// TwinCAT 3 PLC project Core
// ProgramVersion: 3.1.4023.0
// libraries:
//   CmpBitmapPool, * (System)
//   Tc2_MC2, * (Beckhoff Automation GmbH)
//   Tc2_MDP, * (Beckhoff Automation GmbH)
//   Tc2_Standard, * (Beckhoff Automation GmbH)
//   Tc2_System, * (Beckhoff Automation GmbH)
//   Tc2_Utilities, * (Beckhoff Automation GmbH)
//   Tc3_IotBase, * (Beckhoff Automation GmbH)
//   Tc3_Module, * (Beckhoff Automation GmbH)
//   VisuDialogs, * (System)
// project tree:
//   DUTs/ E_Balise.TcDUT, E_Type_motion.TcDUT, E_Type_Tache.TcDUT, ST_Dynamixel_Control_Input.TcDUT, ST_Dynamixel_Control_Output.TcDUT, ST_Tableau.TcDUT
//   / GlobalTextList.TcGTLO
//   GVLs/Action/ G_CAM.TcGVL, G_DXL.TcGVL
//   GVLs/Interruption/ G_Balise.TcGVL
//   GVLs/IO/ G_IO.TcGVL
//   GVLs/Motion/ G_Moteurs.TcGVL, G_Odometrie.TcGVL
//   GVLs/Raspberry PI/ G_RPI.TcGVL
//   GVLs/Structure/ G_EndMatch.TcGVL, G_init.TcGVL, G_Match.TcGVL, G_PreMatch.TcGVL
//   GVLs/Visu/ G_Visus.TcGVL
//   POUs/Action/Camera OAK-D/ FB_CAM.TcPOU, P_cam_launch_pyscript.TcPOU
//   POUs/Action/Dynamixel/ FB_DXL_AX12A.TcPOU, FB_DXL_XL.TcPOU, P_Connect_DXL.TcPOU, P_DXL_launch_pyscript.TcPOU
//   POUs/Action/ ITAction.TcPOU
//   POUs/Communication/ ITCommunication.TcPOU, MQTT.TcPOU
//   POUs/Interruption/ FB_Balise.TcPOU, FB_Timeout.TcPOU, ITInterruption.TcPOU
//   POUs/ MAIN.TcPOU
//   POUs/Motion/ FB_Motion_Odometrie.TcPOU, ITMotion.TcPOU
//   POUs/Structure/Actions/ F_DXL_Position.TcPOU, F_DXL_Reset.TcPOU
//   POUs/Structure/ Structure_MAIN.TcPOU
//   POUs/Structure/Tableaux %28parcours%29/ P_Tableau_Strategie_1.TcPOU (not stored), P_Tableau_Strategie_2.TcPOU (not stored)
//   POUs/Utillity/Debug/ pass.TcPOU (not stored)
//   POUs/Utillity/Logic/ plusOuMoins.TcPOU
//   POUs/Utillity/Maths/ DEGRE2RAD.TcPOU, HYP.TcPOU, RAD2DEGRE.TcPOU
//   POUs/Utillity/Structure/Action/ FinishAction.TcPOU, Next.TcPOU (not stored), StartAction.TcPOU (not stored)
//   POUs/Utillity/Structure/Tableau/ AddStep.TcPOU, EtapeEnCours.TcPOU (not stored), PointsRestants.TcPOU, ReplaceStep.TcPOU
//   POUs/Utillity/Temporisation/ delay.TcPOU
//   TASKs/ BaliseTask.TcTTO, MotionTask.TcTTO, PlcTask.TcTTO, VISU_TASK.TcTTO
//   VISUs/Visu pour debug/ V_Balise.TcVIS, V_Config.TcVIS, V_Deplacement.TcVIS, V_Test.TcVIS
//   VISUs/Images/ ImagePool.TcIPO (not stored)
//   VISUs/Visu pour match/ V_Fin_Match.TcVIS, V_Init.TcVIS, V_Match.TcVIS
//   VISUs/ VisualizationManager.TcVMO (not stored), V_Menu.TcVIS
// real-time tasks:
//   TASK PlcTask: cycle T#10ms, priority 20, ADS port 350
//   TASK VisuTask: cycle T#100000us, priority 30, ADS port 351
//   TASK BaliseTask: cycle T#1ms, priority 5, ADS port 352
//   TASK MotionTask: cycle T#5ms, priority 15, ADS port 353
// motion (NC):
//   TASK NC-Task 1 SAF: cycle T#1ms, priority 4, ADS port 501
//   TASK NC-Task 1 SVB: cycle T#5ms, priority 8, ADS port 511
//   AXIS MoteurG (id 1)
//     Dynamic: Acceleration=3000, Deceleration=3000, Jerk=9000, MaxPosDeviationAuxAxis=5
//     Velo: SlowManual=200
//     PositionAreaControl: Range=10
//     TargetPosControl: Range=10
//     OtherSettings: AllowMotionCmdToSlave=true
//     encoder EncType=4
//       EncPara: ScaleFactorNumerator=162, ScaleFactorDenominator=12800, MaxCount=#x0000ffff
//         ActPosCorrection: Enable=true
//         Inc: RefSoftSyncMask=#x0000ffff
//     drive DrvType=24
//       Analog: VeloReferenz=1700, TorqueSetpointScale=10, ScaleFactorActTorque=0.1
//       TimeComp: TaskDelayCycles=1
//     controller CtrType=1
//       CtrPara: PriorControlFactor=1
//         PosDiffControl: Enable=false, Range=20
//         Observer: BandWidth=20
//   AXIS EncodeurG (id 3)
//     OtherSettings: AllowMotionCmdToSlave=true
//     encoder EncType=4
//       EncPara: ScaleFactorNumerator=162, ScaleFactorDenominator=4096, MaxCount=#x0000ffff
//         Inc: RefSoftSyncMask=#x0000ffff
//     drive DrvType=5
//       Analog: TorqueSetpointScale=10, ScaleFactorActTorque=0.1
//       TimeComp: TaskDelayCycles=1
//     controller CtrType=1
//       CtrPara: PriorControlFactor=1
//         Observer: BandWidth=20
//   AXIS MoteurD (id 2)
//     Dynamic: Acceleration=3000, Deceleration=3000, Jerk=9000, MaxPosDeviationAuxAxis=5
//     Velo: SlowManual=200
//     PositionAreaControl: Range=10
//     TargetPosControl: Range=10
//     OtherSettings: AllowMotionCmdToSlave=true
//     encoder EncType=4
//       EncPara: ScaleFactorNumerator=162, ScaleFactorDenominator=12800, MaxCount=#x0000ffff
//         Inc: RefSoftSyncMask=#x0000ffff
//     drive DrvType=24
//       Analog: VeloReferenz=1700, TorqueSetpointScale=10, ScaleFactorActTorque=0.1
//       TimeComp: TaskDelayCycles=1
//     controller CtrType=1
//       CtrPara: PriorControlFactor=1
//         PosDiffControl: Enable=false, Range=20
//         Observer: BandWidth=20
//   AXIS EncodeurD (id 4)
//     OtherSettings: AllowMotionCmdToSlave=true
//     encoder EncType=4
//       EncPara: ScaleFactorNumerator=162, ScaleFactorDenominator=4096, MaxCount=#x0000ffff
//         Inc: RefSoftSyncMask=#x0000ffff
//     drive DrvType=5
//       Analog: TorqueSetpointScale=10, ScaleFactorActTorque=0.1
//       TimeComp: TaskDelayCycles=1
//     controller CtrType=1
//       CtrPara: PriorControlFactor=1
//         Observer: BandWidth=20
// I/O:
//   DEVICE Device 3 (EtherCAT), AmsNetId 172.16.0.209.4.1
//     Term 1 (EK1100) [EK1100 EtherCAT Coupler (2A E-Bus)]
//       T_Balise (EL1252) [EL1252 2Ch. Fast Dig. Input 24V, 1µs, DC Latch]
//       T_Input (EL1104) [EL1104 4Ch. Dig. Input 24V, 3ms, Sensor Power]
//       T_MoteurG (EL7037) [EL7037 1Ch. Stepper motor output stage (24V, 1.5A)]
//       T_MoteurD (EL7037) [EL7037 1Ch. Stepper motor output stage (24V, 1.5A)]
//       T_Output (EL2798) [EL2798 8Ch. Dig. Output 24V AC/DC, 2A, potential-free]
//       Term 5 (EL9011) [EL9011 End Terminal]
// variable links:
//   NC-Task 1 SAF/Axes/EncodeurD <-> Device 3 (EtherCAT)/Term 1 (EK1100)/T_MoteurD (EL7037)
//     Enc/Inputs/In/nDataIn1 <-> STM External position/External position
//     Enc/Inputs/In/nState4 @bit 1 <-> WcState/InputToggle
//     Enc/Inputs/In/nState4 <-> WcState/WcState
//   NC-Task 1 SAF/Axes/EncodeurG <-> Device 3 (EtherCAT)/Term 1 (EK1100)/T_MoteurG (EL7037)
//     Enc/Inputs/In/nDataIn1 <-> STM External position/External position
//     Enc/Inputs/In/nState4 @bit 1 <-> WcState/InputToggle
//     Enc/Inputs/In/nState4 <-> WcState/WcState
//   NC-Task 1 SAF/Axes/MoteurD <-> Device 3 (EtherCAT)/Term 1 (EK1100)/T_MoteurD (EL7037)
//     Drive/Inputs/In/nState1 @bit 3 <-> STM Status/Error
//     Drive/Inputs/In/nState1 @bit 7 <-> STM Status/Motor stall
//     Drive/Inputs/In/nState1 @bit 5 <-> STM Status/Moving negative
//     Drive/Inputs/In/nState1 @bit 4 <-> STM Status/Moving positive
//     Drive/Inputs/In/nState1 @bit 1 <-> STM Status/Ready
//     Drive/Inputs/In/nState1 <-> STM Status/Ready to enable
//     Drive/Inputs/In/nState1 @bit 6 <-> STM Status/Torque reduced
//     Drive/Inputs/In/nState1 @bit 2 <-> STM Status/Warning
//     Drive/Inputs/In/nState2 @bit 3 <-> STM Status/Digital input 1
//     Drive/Inputs/In/nState2 @bit 4 <-> STM Status/Digital input 2
//     Drive/Inputs/In/nState2 @bit 5 <-> STM Status/Sync error
//     Drive/Inputs/In/nState2 @bit 7 <-> STM Status/TxPDO Toggle
//     Drive/Inputs/In/nState4 @bit 1 <-> WcState/InputToggle
//     Drive/Inputs/In/nState4 <-> WcState/WcState
//     Drive/Outputs/Out/nCtrl1 <-> STM Control/Enable
//     Drive/Outputs/Out/nCtrl1 @bit 2 <-> STM Control/Reduce torque
//     Drive/Outputs/Out/nCtrl1 @bit 1 <-> STM Control/Reset
//     Drive/Outputs/Out/nCtrl2 @bit 3 <-> STM Control/Digital output 1
//     Drive/Outputs/Out/nDataOut2[0] <-> STM Velocity/Velocity
//     Enc/Inputs/In/nDataIn1[0] <-> ENC Status compact/Counter value
//     Enc/Inputs/In/nDataIn2[0] <-> ENC Status compact/Latch value
//     Enc/Inputs/In/nState1 @bit 4 <-> ENC Status compact/Counter overflow
//     Enc/Inputs/In/nState1 @bit 3 <-> ENC Status compact/Counter underflow
//     Enc/Inputs/In/nState1 @bit 7 <-> ENC Status compact/Extrapolation stall
//     Enc/Inputs/In/nState1 <-> ENC Status compact/Latch C valid
//     Enc/Inputs/In/nState1 @bit 1 <-> ENC Status compact/Latch extern valid
//     Enc/Inputs/In/nState1 @bit 2 <-> ENC Status compact/Set counter done
//     Enc/Inputs/In/nState2 @bit 4 <-> ENC Status compact/Status of extern latch
//     Enc/Inputs/In/nState2 <-> ENC Status compact/Status of input A
//     Enc/Inputs/In/nState2 @bit 1 <-> ENC Status compact/Status of input B
//     Enc/Inputs/In/nState2 @bit 2 <-> ENC Status compact/Status of input C
//     Enc/Inputs/In/nState2 @bit 5 <-> ENC Status compact/Sync error
//     Enc/Inputs/In/nState2 @bit 7 <-> ENC Status compact/TxPDO Toggle
//     Enc/Inputs/In/nState4 @bit 1 <-> WcState/InputToggle
//     Enc/Inputs/In/nState4 <-> WcState/WcState
//     Enc/Outputs/Out/nCtrl1 <-> ENC Control compact/Enable latch C
//     Enc/Outputs/Out/nCtrl1 @bit 3 <-> ENC Control compact/Enable latch extern on negative edge
//     Enc/Outputs/Out/nCtrl1 @bit 1 <-> ENC Control compact/Enable latch extern on positive edge
//     Enc/Outputs/Out/nCtrl1 @bit 2 <-> ENC Control compact/Set counter
//     Enc/Outputs/Out/nDataOut1[0] <-> ENC Control compact/Set counter value
//   NC-Task 1 SAF/Axes/MoteurG <-> Device 3 (EtherCAT)/Term 1 (EK1100)/T_MoteurG (EL7037)
//     Drive/Inputs/In/nState1 @bit 3 <-> STM Status/Error
//     Drive/Inputs/In/nState1 @bit 7 <-> STM Status/Motor stall
//     Drive/Inputs/In/nState1 @bit 5 <-> STM Status/Moving negative
//     Drive/Inputs/In/nState1 @bit 4 <-> STM Status/Moving positive
//     Drive/Inputs/In/nState1 @bit 1 <-> STM Status/Ready
//     Drive/Inputs/In/nState1 <-> STM Status/Ready to enable
//     Drive/Inputs/In/nState1 @bit 6 <-> STM Status/Torque reduced
//     Drive/Inputs/In/nState1 @bit 2 <-> STM Status/Warning
//     Drive/Inputs/In/nState2 @bit 3 <-> STM Status/Digital input 1
//     Drive/Inputs/In/nState2 @bit 4 <-> STM Status/Digital input 2
//     Drive/Inputs/In/nState2 @bit 5 <-> STM Status/Sync error
//     Drive/Inputs/In/nState2 @bit 7 <-> STM Status/TxPDO Toggle
//     Drive/Inputs/In/nState4 @bit 1 <-> WcState/InputToggle
//     Drive/Inputs/In/nState4 <-> WcState/WcState
//     Drive/Outputs/Out/nCtrl1 <-> STM Control/Enable
//     Drive/Outputs/Out/nCtrl1 @bit 2 <-> STM Control/Reduce torque
//     Drive/Outputs/Out/nCtrl1 @bit 1 <-> STM Control/Reset
//     Drive/Outputs/Out/nCtrl2 @bit 3 <-> STM Control/Digital output 1
//     Drive/Outputs/Out/nDataOut2[0] <-> STM Velocity/Velocity
//     Enc/Inputs/In/nDataIn1[0] <-> ENC Status compact/Counter value
//     Enc/Inputs/In/nDataIn2[0] <-> ENC Status compact/Latch value
//     Enc/Inputs/In/nState1 @bit 4 <-> ENC Status compact/Counter overflow
//     Enc/Inputs/In/nState1 @bit 3 <-> ENC Status compact/Counter underflow
//     Enc/Inputs/In/nState1 @bit 7 <-> ENC Status compact/Extrapolation stall
//     Enc/Inputs/In/nState1 <-> ENC Status compact/Latch C valid
//     Enc/Inputs/In/nState1 @bit 1 <-> ENC Status compact/Latch extern valid
//     Enc/Inputs/In/nState1 @bit 2 <-> ENC Status compact/Set counter done
//     Enc/Inputs/In/nState2 @bit 4 <-> ENC Status compact/Status of extern latch
//     Enc/Inputs/In/nState2 <-> ENC Status compact/Status of input A
//     Enc/Inputs/In/nState2 @bit 1 <-> ENC Status compact/Status of input B
//     Enc/Inputs/In/nState2 @bit 2 <-> ENC Status compact/Status of input C
//     Enc/Inputs/In/nState2 @bit 5 <-> ENC Status compact/Sync error
//     Enc/Inputs/In/nState2 @bit 7 <-> ENC Status compact/TxPDO Toggle
//     Enc/Inputs/In/nState4 @bit 1 <-> WcState/InputToggle
//     Enc/Inputs/In/nState4 <-> WcState/WcState
//     Enc/Outputs/Out/nCtrl1 <-> ENC Control compact/Enable latch C
//     Enc/Outputs/Out/nCtrl1 @bit 3 <-> ENC Control compact/Enable latch extern on negative edge
//     Enc/Outputs/Out/nCtrl1 @bit 1 <-> ENC Control compact/Enable latch extern on positive edge
//     Enc/Outputs/Out/nCtrl1 @bit 2 <-> ENC Control compact/Set counter
//     Enc/Outputs/Out/nDataOut1[0] <-> ENC Control compact/Set counter value
//   Core/Core Instance <-> Device 3 (EtherCAT)/Term 1 (EK1100)/T_Balise (EL1252)
//     BaliseTask Inputs/G_Balise.Inductif <-> Channel 1/Input
//     BaliseTask Inputs/G_Balise.Laser <-> Channel 2/Input
//     BaliseTask Inputs/ITInterruption.balise.DebutDetection <-> Latch/LatchNeg2
//     BaliseTask Inputs/ITInterruption.balise.DebutTour <-> Latch/LatchPos1
//     BaliseTask Inputs/ITInterruption.balise.FinDetection <-> Latch/LatchPos2
//   Core/Core Instance <-> Device 3 (EtherCAT)/Term 1 (EK1100)/T_Input (EL1104)
//     BaliseTask Inputs/G_IO.bAU <-> Channel 1/Input
//     PlcTask Inputs/G_IO.bCaptDepart <-> Channel 2/Input
//   Core/Core Instance <-> Device 3 (EtherCAT)/Term 1 (EK1100)/T_Output (EL2798)
//     BaliseTask Outputs/G_IO.bMoteurBalise <-> Channel 1/Output
//     PlcTask Outputs/G_IO.bLEDInit <-> Channel 2/Output
//   Core/Core Instance <-> NC-Task 1 SAF/Axes/EncodeurD
//     BaliseTask Inputs/G_Moteurs.axEncodeurD.NcToPlc <-> Outputs/ToPlc
//     MotionTask Outputs/G_Moteurs.axEncodeurD.PlcToNc <-> Inputs/FromPlc
//   Core/Core Instance <-> NC-Task 1 SAF/Axes/EncodeurG
//     MotionTask Inputs/G_Moteurs.axEncodeurG.NcToPlc <-> Outputs/ToPlc
//     MotionTask Outputs/G_Moteurs.axEncodeurG.PlcToNc <-> Inputs/FromPlc
//   Core/Core Instance <-> NC-Task 1 SAF/Axes/MoteurD
//     MotionTask Inputs/G_Moteurs.axMoteurD.NcToPlc <-> Outputs/ToPlc
//     MotionTask Outputs/G_Moteurs.axMoteurD.PlcToNc <-> Inputs/FromPlc
//   Core/Core Instance <-> NC-Task 1 SAF/Axes/MoteurG
//     MotionTask Inputs/G_Moteurs.axMoteurG.NcToPlc <-> Outputs/ToPlc
//     MotionTask Outputs/G_Moteurs.axMoteurG.PlcToNc <-> Inputs/FromPlc

CONFIGURATION Core
    RESOURCE PLC ON TwinCAT3
        TASK BaliseTask(INTERVAL := T#1ms, PRIORITY := 5);
        TASK MotionTask(INTERVAL := T#5ms, PRIORITY := 15);
        TASK PlcTask(INTERVAL := T#10ms, PRIORITY := 20);
        TASK VISU_TASK(INTERVAL := T#100000us, PRIORITY := 30);
        PROGRAM ITInterruption WITH BaliseTask : ITInterruption;
        PROGRAM ITMotion WITH MotionTask : ITMotion;
        PROGRAM MAIN WITH PlcTask : MAIN;
        PROGRAM VisuElems_Visu_Prg WITH VISU_TASK : VisuElems.Visu_Prg;
    END_RESOURCE
END_CONFIGURATION

// ---- DUTs/E_Balise.TcDUT
{attribute 'qualified_only'}
{attribute 'strict'}
TYPE E_Balise :
(
	Angle, Distance
);
END_TYPE

// ---- DUTs/E_Type_motion.TcDUT
TYPE E_Type_motion :
(
	eCoordonne, eMarcheArriereCoordonne, eDistance, eAngle, eCourbe 
);
END_TYPE

// ---- DUTs/E_Type_Tache.TcDUT
TYPE E_Type_Tache :	// Appel des différentes tâches que le robot va faire
(
	eAttendre, eDeplacement, eAction, eFinParcours, eChangementTache
);
END_TYPE

// ---- DUTs/ST_Dynamixel_Control_Input.TcDUT
TYPE ST_Dynamixel_Control_Input :
	STRUCT	
		TypeAX : FB_DXL_AX12A;
		TypeXL : FB_DXL_XL;
		
		bEnableTorque : BOOL;
		bDisableTorque: BOOL;
		
		bLedOn : BOOL;
		IbLedOff : BOOL;
		
		bOperatingMode : BOOL;
		
		bPosition : BOOL;
		bStopPosition : BOOL;
		bResetPosition : BOOL;
		bAcceleration : BOOL;
		bVelocity : BOOL;
		
		ParamOperatingMode_string : STRING;
		ParamReset_BOOL : BOOL;
		ParamPosition_DINT : DINT;
		ParamSpeed_INT : INT;
		ParamAcceleration_USINT : USINT;
		
		bGetLoad : BOOL;
		bGetMovement : BOOL;
		bGetPosition : BOOL;
	END_STRUCT
END_TYPE

// ---- DUTs/ST_Dynamixel_Control_Output.TcDUT
TYPE ST_Dynamixel_Control_Output :
	STRUCT	
		bEnableTorque : BOOL;
		bDisableTorque: BOOL;
		
		bLedOn : BOOL;
		bLedOff : BOOL;
		
		bOperatingMode : BOOL;
		
		bPosition : BOOL;
		bStopPosition : BOOL;
		bResetPosition : BOOL;
		bAcceleration : BOOL;
		bVelocity : BOOL;

		INFO_load_int :INT := -9000;
		INFO_Mouvement_bool : BOOL := 1;
		INFO_Position_dint : DINT := -9000;
	END_STRUCT
END_TYPE

// ---- DUTs/ST_Tableau.TcDUT
TYPE ST_Tableau : // Appel des variables qui permettent de faire les différentes tâches
	STRUCT
		NomEtape			: STRING(50);			// Nom de l'étape en cours => permet de faire des saut dans le tableau pour cibler une action en particulier
		EtapeCible			: STRING(50); 			// Nom de l'étape à laquelle on veut aller
		TypeTache			: E_Type_Tache;			// Permet la tâche qu'on va faire à la ligne du tableau
		TypeDeplacement     : E_Type_motion;        // Permet de choisir le type de déplacement
		TypeAction			: STRING(50);			// Choisi le type d'action
		lrPositionX_mm		: LREAL;				// Position en x que l'on veut donner au robot lors d'un déplacement
		lrPositionY_mm		: LREAL;				// Position en y que le robot doit atteindre lors d'un déplacement
		lrAngleVoulu_deg	: LREAL;				// Angle que l'on veut atteindre lors d'une rotation, en fonction de l'angle de référence dans Odometrie
		lrDistanceVoulu_mm	: LREAL;				// Distance que le robot va avancer
		lrVitesse_mms		: LREAL;				// Vitesse de déplacement du robot quand il fait un mouvement ou une rotation
		lrRayonCourbe_mm	: LREAL;
		tAttente_ms			: TIME;					// Temps que le robot va attendre quand la tâche attente est choisie
		uiAjoutPoints_pts	: INT;					// Nombre de points que l'on veut ajouter sur le compteur
		bArretDetection		: BOOL;					// Désactivation de la détection de la balise, le robot ne s'arrête plus quand il détecte un adversaire, sert à pouvoir démarrer si nos robots ont aussi des catadioptres
	END_STRUCT
END_TYPE

// ---- GVLs/Action/G_CAM.TcGVL
{attribute 'qualified_only'}
//author: Alec Horth

// servent à la communication PYADS (! ne pas modifier)
//seulement accessible au FB "FB_CAM"
VAR_GLOBAL
	//RUN variable => active les fonctionnalités de la caméra
	//sinon les fonctions ne sont pas active pour economiser les ressources de la CPU (!! garde la dernière valeur)
	RUN_STEREO			:BOOL; //mesure de proximité
	RUN_ARUCO			:BOOL; //liste les ID des tags aruco présents dans le champ de vision de la caméra
	
	//retour de la caméra 
	proximite			:USINT; //mesure de proximité de 0 à 3 
							   //(0:champ de vision vide, 1:objet détecté, 2:object proche, 3:distance critique)
	tag_aruco			:ARRAY[0..10] OF INT; //list les id des tags aruco présent 
											  // max 10 tag détectés en même temps (défini par la longeur max de la liste)
	taille_tag_aruco_cm :INT;
	ID_tag_aruco		:INT;
	
	//fonctions du script python
	STOP_PYSCRIPT		:BOOL; //arrête le script python
	restart_py_script	:BOOL:= FALSE; //démarre le script python
	bPyscript_running	:BOOL;		//le script python est actif
END_VAR

// ---- GVLs/Action/G_DXL.TcGVL
{attribute 'qualified_only'}
//author: Alec Horth

//servent à la communication PYADS (! ne pas modifier)
//seulement accessible au FB "FB_DXL_ALL"
VAR_GLOBAL 
	//activation des fonction du moteur dynamixel
	bRun					:BOOL;		// action la fonction
	bStop_python_script		:BOOL; 		// arrête le script python
	
	//commande envoyé au moteur 
	iID						:INT;		// id du motor 
	usiMotor_type			:USINT;		// type du moteur 1 => AX12A, 2 => XL430
	usiFonction 			:USINT;		// fonction à executer
	sMode					:STRING;	// configuration du mode de fonctionnement (position, velocité)
	iSpeed					:INT;		// configuration de la vitesse
	diPosition				:DINT;		// configuration de la position
	usiAcceleration			:USINT; 	// configuration de l'accelération du moteur
	bReset					:BOOL;		// reset de la position en mode multitour
	
	//information du moteur
	iDxl_load				:INT; 
	diDxl_position			:DINT;
	bDxl_movement			:BOOL;
	bDone					:BOOL;		//action reçue et envoyée
	bPyscript_running		:BOOL;		//le script python est actif
	
	// semaphore (contrôle qu'il n'y aie qu'une communication à la fois avec le moteur)
	// indique l'ID de l'instance qui a le droit de communiquer avec le moteur
	// Token disponible => -16#FE ou -254 ou -1 * id_du_moteur_ayant_la_permission
	bToken					:INT:= -16#FE; 
	
	//activation du script python
	bRestart_py_script		:BOOL;
END_VAR

//type de commandes à envoyer au moteur
VAR_GLOBAL CONSTANT 
	//RAM
	usiOPERATING_MODE		:USINT := 0;
	
	//ACTION
	usiENABLE_TORQUE		:USINT := 1; 
	usiDISABLE_TORQUE		:USINT := 2;
	usiLED_ON				:USINT := 3;
	usiLED_OFF				:USINT := 4;
	usiGOAL_ACCELERATION	:USINT := 5;
	usiGOAL_VELOCITY		:USINT := 6;
	usiGOAL_POSITION		:USINT := 7;
	
	//prédicat
	usiGET_PRESENT_POSITION:USINT := 8;
    usiGET_PRESENT_LOAD	:USINT := 9;
    usiGET_PRESENT_MOVEMENT:USINT := 10;
	
	//fonction accessoire du mode position
	usiSTOP_POSITION		:USINT := 11;
	usiRESET_POSITION		:USINT := 12;
	
	//token libre
	iOPEN_TOKEN			:INT   := -254;
END_VAR

// ---- GVLs/Interruption/G_Balise.TcGVL
{attribute 'qualified_only'}
VAR_GLOBAL
	Laser 				AT%I* 	: BOOL; 			//capteur optique de proximité (avec le mirroir)
	Inductif 			AT%I* 	: BOOL; 			//capteur induction sous la balise	
	
	iNombreEnnemi 				: INT;				// nombre de fronts montants du laser, nombres d'ennemis détectés en un tour
	ArrayEnnemi					: ARRAY [0..2,0..1] OF LREAL; 	// 	colonnes = ennemis 	[colonne, ligne]
																//	ligne 0 = Angle 	[colonne, ligne]
                                                        		// 	ligne 1 = Distance 	[colonne, ligne]
	
	bFront 						: BOOL;				//adversaire devant
	bBack 						: BOOL;				//adversaire derrière
	bLeft						: BOOL;				//adversaire à gauche
	bRight						: BOOL;				//adversaire à droite
	bProche						: BOOL;				//obstacle détecté proche
	bClose 						: BOOL;				//obstacle détecté vraiment proche	
	
	lrDistance_1				: LREAL;			// Distance du premier ennemi détecté, est envoyée dans la visu balise
	lrDistance_2				: LREAL;			// Distance du deuxième adversaire détecté, est envoyée dans la visu balise
	lrDistance_3				: LREAL;			// Distance du troisième ennemi détecté, est envoyée dans la visu balise
	lrAngle_1					: LREAL;			// Angle auquel le premier ennemi est détecté pour pouvoir le voir dans la visu balise
	lrAngle_2					: LREAL;			// Angle de détection du deuxième adversaire, l'angle est envoyé dans la visu balise
	lrAngle_3					: LREAL;			// Angle du troisième adversaire , permet de savoir la position de l'ennemi dans la visu balise

	lrCoord_X1					: LREAL;			//coordonné X de l'enemi 1 selon le système de l'odométrie (activé avec la visu)
	lrCoord_Y1					: LREAL;			//coordonné Y de l'enemi 1 selon le système de l'odométrie (activé avec la visu)
	lrCoord_X2					: LREAL; 			//coordonné X de l'enemi 2 selon le système de l'odométrie (activé avec la visu)
	lrCoord_Y2					: LREAL; 			//coordonné Y de l'enemi 2 selon le système de l'odométrie (activé avec la visu)
	lrCoord_X3					: LREAL;			//coordonné X de l'enemi 3 selon le système de l'odométrie (activé avec la visu)
	lrCoord_Y3					: LREAL;			//coordonné Y de l'enemi 3 selon le système de l'odométrie (activé avec la visu)
END_VAR

// ---- GVLs/IO/G_IO.TcGVL
{attribute 'qualified_only'}
VAR_GLOBAL
	// Variable en cas de panneau de commande sur le robot, sinon remplacer par des boutons visus.
	bAU				AT%I*: BOOL;	// Bouton d'arrêt d'urgence, contact NC
	bChoixCote		AT%I*: BOOL;	// Selecteur deux positions pour le choix du coté de départ (jaune=true, violet=false)
	bInitRobot		AT%I*: BOOL;	// Bouton poussoir pour l'initialisation du robot, action et position
	bCaptDepart		AT%I*: BOOL;	// Capteur inductif pour commencer un match
	bReset			AT%I*: BOOL;	// Redémarre Twincat
	
	bLEDInit		AT%Q*: BOOL;	// LED robot initialisé, s'allume quand le robot est initialisé
	bMoteurBalise	AT%Q*: BOOL;	// Moteur de la balise, fait tourner le rayon pour détecter les adversaires
END_VAR

// ---- GVLs/Motion/G_Moteurs.TcGVL
{attribute 'qualified_only'}
VAR_GLOBAL
	axMoteurG		: AXIS_REF;			// Moteur gauche de la base roulante
	axMoteurD		: AXIS_REF;			// Moteur droit de la base roulante
	axEncodeurG		: AXIS_REF;			// Encodeur gauche de la base roulante, permet de savoir les déplacements sur la table
	axEncodeurD		: AXIS_REF;			// Encodeur droit de la base roulante, permet de connaitre les déplacements sur la table
	
	mcPowerG		: MC_Power;			// Bloc MC_Power, alimente le moteur gauche de la base roulante 
	mcPowerD		: MC_Power;			// Bloc MC_Power, alimente le moteur droite de la base roulante
	
	mcRelativeD		: MC_MoveRelative;	// Bloc move relative du moteur gauche, permet au robot de se déplacer en fonction de sa position
	mcRelativeG		: MC_MoveRelative;	// Bloc move relative du moteur droit, permet au robot de se déplacer en fonction de sa position
	
	mcSuperPosD		: MC_MoveSuperImposed;
	mcSuperPosG		: MC_MoveSuperImposed;
										// Blocs d'arrêts (pause) des moteurs des roues de la base roulante
	mcHaltDroite 	: MC_Halt;			//Arrêt moteur droit
	mcHaltGauche 	: MC_Halt;			//Arrêt moteur gauche
	
	mcResetGau		: MC_Reset;			// Bloc de reset du moteur gauche de la base roulante
	mcResetDro		: MC_Reset;			// Bloc qui réinitialise le moteur droit de la base roulante
	
	mcStopG			: MC_Stop;			// Bloc stop du moteur gauche, arrête le moteur gauche de la base roulante
	mcStopD			: MC_Stop;			// Bloc stop du moteur droit, arrête le moteur droit de la base roulante
END_VAR

// ---- GVLs/Motion/G_Odometrie.TcGVL
{attribute 'qualified_only'}
VAR_GLOBAL
	// positions actuelles du robot
	lrAngle				: LREAL;	// Angle de la position du robot en radians, à l'angle 0, le robot fait face au long côté
	lrAngleDeg			: LREAL;	// Angle de la position du robot en degrés 
	lrPositionX			: LREAL;	// Position en X du robot sur la table (sens 3m)
	lrPositionY			: LREAL;	// Position en Y du robot sur la table (sens 2m)
END_VAR

// ---- GVLs/Raspberry PI/G_RPI.TcGVL
{attribute 'qualified_only'}
VAR_GLOBAL
	//Grille d'où sont passé les robots adverses
	grid : ARRAY [0..5] OF ARRAY [0..8] OF BOOL;
	//Reset de la grille dans le raspberry pi
	reset : BOOL;
END_VAR

// ---- GVLs/Structure/G_EndMatch.TcGVL
{attribute 'qualified_only'}
VAR_GLOBAL
	icounter : INT;
	bShutdown_done : BOOL;
END_VAR

// ---- GVLs/Structure/G_init.TcGVL
{attribute 'qualified_only'}
VAR_GLOBAL
	ietapeInit    	:INT;
	binitDone 		:BOOL;
	icounter 		:INT;
	iNombreEtapeInit:INT;
END_VAR

// ---- GVLs/Structure/G_Match.TcGVL
{attribute 'qualified_only'}
VAR_GLOBAL
	TimeStartLigne  	: TIME;
	TimeStartMatch 		: TIME;
	TimeMatch 			: TIME;
	PointMatch 			: LREAL;
	MatchEnCours		: BOOL;
	RetourEnCours		: BOOL;

	Tableau 			: ARRAY[0..100] OF ST_Tableau;
	iLigne 				: INT;
	NextLigne			: BOOL;
	iCounter			: INT;
	
	bExecuteDeplacement : BOOL;
	bDeplacementFini	: BOOL;
	bActionFinie		: BOOL;
	
	iEtapeAction 		: INT;
	iAsyncAction 		: STRING; 
END_VAR

// ---- GVLs/Structure/G_PreMatch.TcGVL
{attribute 'qualified_only'}
VAR_GLOBAL
	bPrematchActive : BOOL;
END_VAR

// ---- GVLs/Visu/G_Visus.TcGVL
{attribute 'qualified_only'}
VAR_GLOBAL
	//Visu V_Config
	bConfigEnable : BOOL;	
	
	//indicateurs
	bConfigMoteurReady	: BOOL;
	bConfigReady : BOOL;
	bConfigMoveDone : BOOL;
	
	//Bouton 
	bConfigStart : BOOL;
	bConfigReset : BOOL;
	bConfigBalise : BOOL;
	bConfigMoteurPower : BOOL;
	bConfigMarcheArriere : BOOL;
	bConfigChoixCote : BOOL; //True = atelier, FALSE = bureau	
	
	//consigne de position et vitesse
	lrConfigPosX : LREAL;
	lrConfigPosY : LREAL;
	lrConfigVitesse : LREAL;
	lrConfigAcc : LREAL;
	lrConfigDecc : LREAL;
	
	//monitoring de la position
	lrConfigErreurX : LREAL;
	lrConfigErreurY : LREAL;
	lrConfigErreurX_pourcent : LREAL;
	lrConfigErreurY_pourcent : LREAL;
	
	//Visu V_Init
	bInitStart		   	: BOOL;
	iInitProgressBar    : INT;
	bInitPrematch		: BOOL;
	bInitChoixCote 		: BOOL;
	iInitChoixParcours 	: INT;
	bInitStartMatch		: BOOL;
	bInitPyScriptRunning: BOOL;
	bInitStartPyscript	: BOOL;
	bInitStopPyscript	: BOOL;
	
	//Visu V_Menu
	bMenuRestart		: BOOL;
	
	//Visu V_Match
	bMatchEnemi			: BOOL;
	
	//Visu V_Test
	bTestEnable			: BOOL;
	sTestFunction1		:STRING(50);
	sTestFunction2		:STRING(50);
	sTestFunction3		:STRING(50);
	sTestFunction4		:STRING(50);
	sTestFunction5		:STRING(50);
	sTestFunction6		:STRING(50);
	
	sTestBouton1		:BOOL;
	sTestBouton2		:BOOL;
	sTestBouton3		:BOOL;
	sTestBouton4		:BOOL;
	sTestBouton5		:BOOL;
	sTestBouton6		:BOOL;
END_VAR

// ---- POUs/Interruption/ITInterruption.TcPOU
PROGRAM ITInterruption
VAR
	//FB qui interrompent un tâche en cours de la structure via des signaux d'interruption - Alec 08.11.23
	balise : FB_Balise;			//gère la Balise et les visus qui lui sont associé 
	timeout: FB_Timeout;		//le temps du match arrive à sa fin
	restartTwincat : TC_Restart;//redémarre twincat
END_VAR

VAR_INPUT
	//interface - Alec 08.11.23
	IbStartBalise 		:BOOL; //Démarre le moteur de la balise
	IbMatchEnCours		:BOOL; //Match en cours
	IbStartVisuBalise	:BOOL; //Démarre la visu balise (à ne pas faire tourner pendant les matchs dans l'idéal car elle demande pas mal de ressource)
	IbRestartTwincat	:BOOL; //Redémarre twincat
	IbArretDetection	:BOOL; //Arrête la détection pendant que la variable est à TRUE
END_VAR

VAR_OUTPUT
	//Signaux d'interruption qui influencent le system - Alec 08.11.23
	QbStopMotion		:BOOL;	//Arrête les moteurs du robot 
	QbPauseMotion  		:BOOL;	//interrompt le déplacement du robot tant que la variable est à TRUE 
	QbResetMotion 		:BOOL;	//Fait un reset des moteurs en cas d'erreur 
	QbEndMatch 			:BOOL;	//Si _3_Match va en _8_EndMatch
	QbAbortTask			:BOOL;	//Arrête la tâche en cours (dépend de l'étape actuel de la structure)
								//si _1_INIT => recommence l'init
								//si _2_PREMATCH => retourne à l'init
								//si _6_INTERRUPTION => change la ligne actuelle du Tableau (changement de tâche)
END_VAR
VAR // added by the converter: edge detectors and wires of the graphical bodies
    _w1, _w2 : BOOL;
END_VAR

// Le capteur de la balise ne détecte pas forcément toute la surface du catadioptre,
// Il faut un peu tester et adapter la valeur uirayonCatadioptre pour que le résultat
// soit plus précis (max 50mm). Vous pouvez utiliser la Visu V_Balise - Alec 08.11.23
balise(
    bstartBalise := IbStartBalise,
    bStopDetection := IbArretDetection,
    uirayonCatadioptre := 35,
    tTimeBeforeAbort := T#5s,
    uiDistanceArretRapide := 700,
    uiDistanceArretLente := 400,
    iVitesseRapide := 500,
    iVitesseLente := 200,
    bactivateVisu := IbStartVisuBalise); // FB_Balise
QbAbortTask := _w1;
_w1 := balise.bAbort OR _w2;
_w2 := NOT IbMatchEnCours AND NOT G_IO.bAU;
QbEndMatch := IbMatchEnCours AND NOT G_IO.bAU;
QbStopMotion := NOT G_IO.bAU;
restartTwincat(RESTART := IbRestartTwincat); // TC_Restart
QbPauseMotion := balise.bStop;
QbResetMotion := NOT G_IO.bAU;

END_PROGRAM

// ---- POUs/Interruption/FB_Balise.TcPOU
FUNCTION_BLOCK FB_Balise
VAR_INPUT
	bstartBalise 			:BOOL; //démarre la balise
	bStopDetection 			:BOOL; //active ou désactive la logique de détection
	uirayonCatadioptre 		:UINT; //rayon détectable du catadioptre [mm]
	tTimeBeforeAbort   		:TIME; //si la balise détect qqch pendant un temps plus long que cette variable, le FB renvoie un 2e signal pour que le robot tente éventuellement un évitement
	
	uiDistanceArretRapide	:UINT; //distance de détection lorsque le robot se déplace à la vitesseRapide [mm]
	uiDistanceArretLente 	:UINT; //distance de détection lorsque le robot se déplace à la vitesseLente [mm]
	iVitesseRapide		 	:INT;  //[mm/s]
	iVitesseLente			:INT;  //[mm/s]
	bactivateVisu     		:BOOL; //active la visu
END_VAR

VAR_OUTPUT
	bStop 					:BOOL; //la balise détect qqch
	bAbort					:BOOL; //si la balise détecte qqch plus longtemps que tTimeBeforeAbort, met la variable à true pour que le robot tente un évitement par exemple
END_VAR

VAR
	past_time 				:TIME; //tempo pour laisser 2s au moteur de la balise avant de commencer la détection
	time_since_enemi_detect :TIME; //temps depuis le début de la détection d'un enemi
	balise_active 			:BOOL; //la balise tourne depuis 2s

	DebutDetection	AT%I*: ULINT;  //Temps depuis le début de la détection 	(Front montant laser)
	FinDetection 	AT%I*: ULINT;  //Temps depuis la fin de la détection 	(Front descendant laser)
	DebutTour 		AT%I*: ULINT;  //Temps depuis le début du tour du laser	(Front montant inductif)
	
	R_EdgeLaser		: R_Trig;	//Front montant du laser
	F_EdgeLaser		: F_Trig;	//Front descendant du laser
	F_EdgeInductif	: F_Trig;	//Front descendant de l'inductif, signifie la fin du tour de la balise
	
//-----------------

	Temps_Tour			:	ULINT;	// Temps d'un tour de la balise
	Temps_Tour_1		:	ULINT;	// Temps d'un tour de la balise
	Temps_Tour_2		:	ULINT;	// Temps d'un tour de la balise
	
	TValeursBrutes		: 	ARRAY [0..2,0..1] OF LREAL;	// Tableau stockant les valeurs des ennemis pour traitement,	colonnes = ennemis
														//																ligne 0 = écart entre référence et fin de détection
                                                        // 																ligne 1 = temps détection
//-----------------
	icounter		: INT;			// valeur boucle for
	PresenceEnnemi 	: ARRAY [0..2] OF BOOL;  
END_VAR

VAR //Pour visu
	posiX1 : LREAL;
	posiY1 : LREAL;
	posiX2 : LREAL;
	posiY2 : LREAL;
	posiX3 : LREAL;
	posiY3 : LREAL;
	
	CoordX1 : LREAL;
	CoordY1 : LREAL;
	CoordX2 : LREAL;
	CoordY2 : LREAL;
	CoordX3 : LREAL;
	CoordY3 : LREAL;
	
	AngleRAD : LREAL;
	AngleRAD2 : LREAL;
	AngleRAD3 : LREAL;
	
	Nothing1 : BOOL ;
	Nothing2 : BOOL ;
	Nothing3 : BOOL ;
	
	Angle0deg : BOOL;
	Angle90deg: BOOL;
	Angle180deg: BOOL;
	Angle270deg: BOOL;
	
	D1_40cm : BOOL;
	D2_40cm : BOOL;
	D3_40cm : BOOL ;
END_VAR;

VAR CONSTANT
	uiDistanceDetectionMax_mm : UINT := 975;
	uiMarge					  : UINT := 20;
END_VAR

//_____________________________________________________________________________________________________________________________________________
//
// Activation de la balise
//______________________________________________________________________________________________________________________________________________

IF bstartBalise THEN 
	G_IO.bMoteurBalise	:= TRUE;
	IF NOT balise_active THEN 
		balise_active := TRUE;
		past_time := TIME();
	END_IF;
ELSE
	balise_active := FALSE;
	G_IO.bMoteurBalise	:= FALSE;
END_IF

//______________________________________________________________________________________________________________________________________________
//
// Gestion et calculs des données de la balise
//______________________________________________________________________________________________________________________________________________

// Si la balise est active depuis 2s
IF balise_active AND delay(past_time, T#2S) THEN 
	//----------------------------------------------------------------------------------------------- DEFINITION DES FRONTS DE LA BALISE ET DE L'INDUCTIF
	F_EdgeLaser	 	(CLK := G_Balise.Laser);		// Début de captation d'un ennemi
	R_EdgeLaser		(CLK := G_Balise.Laser);		// Fin de captation d'un ennemi
	F_EdgeInductif 	(CLK := G_Balise.Inductif);		// Fin d'un tour de la balise
	
	//---------------------------------------------------------------------------------------------------------------- DEFINITION DU NOMBRE DE DETECTIONS
	IF F_EdgeLaser.Q AND (G_Balise.iNombreEnnemi <= 3) THEN	// limitation à max 3 détections
		G_Balise.iNombreEnnemi := G_Balise.iNombreEnnemi + 1;
	END_IF
	
	//--------------------------------------------------------------------------------- DEFINITION DES TEMPS DE DETECTION ET DES ECARTS AVEC LA REFERENCE
	// Quand un ennemi est détecté, les valeurs de temps de détection et de tour sont mise en mémoire, le > 1000000000000 sert à empècher les valeurs trop élevées d'être envoyées dans le programme et à bloquer la valeur précédente
	IF R_EdgeLaser.Q AND (G_Balise.iNombreEnnemi > 0 AND G_Balise.iNombreEnnemi <=3) AND NOT ((FinDetection - DebutTour)> 1000000000000) THEN	
		TValeursBrutes [(G_Balise.iNombreEnnemi - 1),E_Balise.angle] := ULINT_TO_LREAL (FinDetection - DebutTour);		// Inscription durée entre le 0° et la fin de détection de l'ennemi
		TValeursBrutes [(G_Balise.iNombreEnnemi - 1),E_Balise.distance] := ULINT_TO_LREAL (FinDetection - DebutDetection);// Inscription durée détection de l'ennemi
	END_IF
	
	//------------------------------------------------------------------------------------------------------------------------ CALCUL DES VALEURS FINALES
	// durée d'un tour du laser,les 3 valeurs de tours sont chacune décalées d'un cycle automate, pour ne jamais perdre de cycle
	IF NOT (Temps_Tour_2 = DebutTour) THEN;
		Temps_Tour_2 := DebutTour;
	END_IF
	IF NOT (Temps_Tour_1 = Temps_Tour_2) THEN;
		Temps_Tour := Temps_Tour_2 - Temps_Tour_1;
	END_IF
	Temps_Tour_1 := Temps_Tour_2;
	
	//----------------------------------------------------------------
	// A la fin d'un tour, si on détecte au moins un ennemi 
	IF F_EdgeInductif.Q THEN
		// Calcul des angles et distances des ennemis
		IF G_Balise.iNombreEnnemi <> 0 AND G_Balise.iNombreEnnemi <= 3 THEN 
			FOR icounter := 0 TO (G_Balise.iNombreEnnemi - 1) DO
				
				G_Balise.ArrayEnnemi [icounter,E_Balise.angle] := _M_Angle_enemi(//calcule de l'angle de l'enemi
								Time_Tour			:= ULINT_TO_LREAL (Temps_Tour),
							  	Time_FinDetection	:= TValeursBrutes [icounter,E_Balise.Angle],
							  	Time_DetecEnnemi	:= TValeursBrutes [icounter,E_Balise.Distance]);
				
				G_Balise.ArrayEnnemi [icounter,E_Balise.distance] := _M_Distance_enemi(//calcul de la distance de l'enemi
								Time_Tour			:= ULINT_TO_LREAL (Temps_Tour),
							  	Time_FinDetection	:= TValeursBrutes [icounter,E_Balise.Angle],
							  	Time_DetecEnnemi	:= TValeursBrutes [icounter,E_Balise.Distance]);			  
			END_FOR
		END_IF
		
		// Remplissage du reste du tableau si pas 3 détections
		IF  G_Balise.iNombreEnnemi <= 2 AND G_Balise.iNombreEnnemi > 0 THEN
			FOR icounter := 2 TO G_Balise.iNombreEnnemi BY (-1) DO	// écriture de la valeur d'erreur dans le tableau de données brutes
				G_Balise.ArrayEnnemi [icounter, E_Balise.angle] := 9000;
				G_Balise.ArrayEnnemi [icounter, E_Balise.distance] := 9000;
			END_FOR
		ELSIF G_Balise.iNombreEnnemi = 0 THEN
			FOR icounter := 2 TO 0 BY (-1) DO	// écriture de la valeur d'erreur dans le tableau de données brutes
				G_Balise.ArrayEnnemi [icounter, E_Balise.Angle] := 9000;
				G_Balise.ArrayEnnemi [icounter, E_Balise.Distance] := 9000;
			END_FOR
		END_IF
		
		// reset des compteurs et tableaux (sauf données finales) si tour de balise terminé (front descendant inductif)
		G_Balise.iNombreEnnemi := 0;
	END_IF
END_IF


//______________________________________________________________________________________________________________________________________________
//
// Analyse de la position et action sur le system 
//______________________________________________________________________________________________________________________________________________

IF NOT bStopDetection THEN 
	//Détection de présence d'obstacles -----------------------------------------------------------------------------------------------------------------
	
	//Détecteur de présence obstacle dans la portée de détection réglée
	FOR icounter := 0 TO 2 DO
		IF	(G_Balise.ArrayEnnemi[icounter,E_Balise.Distance] < uiDistanceDetectionMax_mm AND G_Balise.ArrayEnnemi[icounter,E_Balise.Distance] <> 0) AND
			(G_Balise.ArrayEnnemi[icounter,E_Balise.Angle] > 0	AND G_Balise.ArrayEnnemi[icounter,E_Balise.Angle] < 360) THEN
			PresenceEnnemi [icounter] := TRUE;
		ELSE
			PresenceEnnemi [icounter] := FALSE;
		END_IF
	END_FOR
	
	//Position des robots adverses (point de vue du robot)------------------------------------------------------------------------------------------------------------------------------------------------------------
	
	//obstacle face avant (entre 90 et 0°)
	
	IF		(PresenceEnnemi [0] AND (G_Balise.ArrayEnnemi [0,E_Balise.Angle]	<= 90+uiMarge AND G_Balise.ArrayEnnemi [0,E_Balise.Angle]	>= 0-uiMarge))
		OR	(PresenceEnnemi [1] AND (G_Balise.ArrayEnnemi [1,E_Balise.Angle]	<= 90+uiMarge AND G_Balise.ArrayEnnemi [1,E_Balise.Angle]	>= 0-uiMarge))
		OR	(PresenceEnnemi [2] AND (G_Balise.ArrayEnnemi [2,E_Balise.Angle]	<= 90+uiMarge AND G_Balise.ArrayEnnemi [2,E_Balise.Angle]	>= 0-uiMarge))	THEN;
		
			G_Balise.bFront := TRUE; //-----------Obstacle confirmé derrière
	ELSE 
			G_Balise.bFront := FALSE;
	END_IF
	
	//obstacle face arrière (entre 270 et 180°)
	IF		(PresenceEnnemi [0] AND (G_Balise.ArrayEnnemi [0,E_Balise.Angle]	<= 270+uiMarge AND G_Balise.ArrayEnnemi [0,E_Balise.Angle]	>= 180-uiMarge)) 
		OR	(PresenceEnnemi [1] AND (G_Balise.ArrayEnnemi [1,E_Balise.Angle]	<= 270+uiMarge AND G_Balise.ArrayEnnemi [1,E_Balise.Angle]	>= 180-uiMarge)) 
		OR	(PresenceEnnemi [2] AND (G_Balise.ArrayEnnemi [2,E_Balise.Angle]	<= 270+uiMarge AND G_Balise.ArrayEnnemi [2,E_Balise.Angle]	>= 180-uiMarge))	THEN;
		
			G_Balise.bBack := TRUE; //-----------Obstacle confirmé devant
	ELSE 
			G_Balise.bBack := FALSE;
	END_IF
	
	//obstacle coté droit (entre 270 et 360°)
	IF		(PresenceEnnemi [0] AND (G_Balise.ArrayEnnemi [0,E_Balise.Angle]	< 360+uiMarge AND G_Balise.ArrayEnnemi [0,E_Balise.Angle]	> 270-uiMarge))
		OR	(PresenceEnnemi [1] AND (G_Balise.ArrayEnnemi [1,E_Balise.Angle]	< 360+uiMarge AND G_Balise.ArrayEnnemi [1,E_Balise.Angle]	> 270-uiMarge))
		OR	(PresenceEnnemi [2] AND (G_Balise.ArrayEnnemi [2,E_Balise.Angle]	< 360+uiMarge AND G_Balise.ArrayEnnemi [2,E_Balise.Angle]	> 270-uiMarge))		THEN;
		
			G_Balise.bRight := TRUE;	//------------ Obstacle confirmé à droite
	ELSE
			G_Balise.bRight := FALSE;
	END_IF
	
	//obstacle coté gauche (entre 180 et 90°)
	IF		(PresenceEnnemi [0] AND (G_Balise.ArrayEnnemi [0,E_Balise.Angle]	< 180+uiMarge AND G_Balise.ArrayEnnemi [0,E_Balise.Angle]	> 90-uiMarge))
		OR	(PresenceEnnemi [1] AND (G_Balise.ArrayEnnemi [1,E_Balise.Angle]	< 180+uiMarge AND G_Balise.ArrayEnnemi [1,E_Balise.Angle]	> 90-uiMarge))
		OR	(PresenceEnnemi [2] AND (G_Balise.ArrayEnnemi [2,E_Balise.Angle]	< 180+uiMarge AND G_Balise.ArrayEnnemi [2,E_Balise.Angle]	> 90-uiMarge))		THEN;
		
			G_Balise.bLeft := TRUE;	//------------ Obstacle confirmé à gauche
	ELSE
			G_Balise.bLeft := FALSE;
	END_IF
	
	//obstacle très près (distance min. sans gêner notre robot, prendre en compte goblets et distance d'arrêt + pinces)
	IF  	(PresenceEnnemi [0] AND G_Balise.ArrayEnnemi[0,E_Balise.Distance]	<= uiDistanceArretLente)
		OR	(PresenceEnnemi [1] AND G_Balise.ArrayEnnemi[1,E_Balise.Distance]	<= uiDistanceArretLente)
		OR	(PresenceEnnemi [2] AND G_Balise.ArrayEnnemi[2,E_Balise.Distance]	<= uiDistanceArretLente) THEN
	
			G_Balise.bClose := TRUE;//-------- Obstacle trop proche
	ELSE
			G_Balise.bClose := FALSE ;
	END_IF
	
	// Obstacle a une distance proche, le robot s'arrête si il va trop vite
	IF  	(PresenceEnnemi [0] AND G_Balise.ArrayEnnemi[0,E_Balise.Distance]	<= uiDistanceArretRapide)
		OR	(PresenceEnnemi [1] AND G_Balise.ArrayEnnemi[1,E_Balise.Distance]	<= uiDistanceArretRapide)
		OR	(PresenceEnnemi [2] AND G_Balise.ArrayEnnemi[2,E_Balise.Distance]	<= uiDistanceArretRapide) THEN
		
			G_Balise.bProche := TRUE;//------- Obstacle proche
	ELSE
			G_Balise.bProche := FALSE;
	END_IF
	
	//Logique d'arrêt------------------------------------------------------------------------------------------------------------------------------------
	IF	(G_Moteurs.mcRelativeD.Distance > 0 AND G_Moteurs.mcRelativeG.Distance > 0 AND	G_Balise.bFront	AND (G_Moteurs.AxEncodeurD.NcToPlc.ActVelo > iVitesseRapide)) OR	// Si le robot avance vite mais qu'il y a un ennemi devant
		(G_Moteurs.mcRelativeD.Distance < 0 AND G_Moteurs.mcRelativeG.Distance < 0 AND	G_Balise.bBack	AND (G_Moteurs.AxEncodeurD.NcToPlc.ActVelo < -iVitesseRapide)) OR	// Si le robot recule vite mais qu'il y a un ennemi derrière
		
		(G_Moteurs.mcRelativeD.Distance > 0 AND G_Moteurs.mcRelativeG.Distance > 0 AND	G_Balise.bFront	AND G_Balise.bProche AND (G_Moteurs.AxEncodeurD.NcToPlc.ActVelo > iVitesseLente)) OR	// Si le robot avance mais qu'il y a un ennemi devant
		(G_Moteurs.mcRelativeD.Distance < 0 AND G_Moteurs.mcRelativeG.Distance < 0 AND	G_Balise.bBack	AND G_Balise.bProche AND (G_Moteurs.AxEncodeurD.NcToPlc.ActVelo < -iVitesseLente)) OR	// Si le robot recule mais qu'il y a un ennemi derrière
		
		(G_Moteurs.mcRelativeD.Distance > 0 AND G_Moteurs.mcRelativeG.Distance > 0 AND	G_Balise.bFront	AND	G_Balise.bClose) OR	// Si le robot avance lentement ou veut avancer mais qu'il y a un ennemi devant
		(G_Moteurs.mcRelativeD.Distance < 0 AND G_Moteurs.mcRelativeG.Distance < 0 AND	G_Balise.bBack 	AND	G_Balise.bClose) OR	// Si le robot recule lentement ou veut reculer mais qu'il y a un ennemi derrière
		
		(G_Balise.bClose) 	THEN	//Si un ennemi nous empêche de tourner
		
		//compte le temps depuis le moment de détection d'un adversaire
		IF NOT bStop THEN 
			time_since_enemi_detect := TIME();
		END_IF
		bStop := TRUE;	// Interruption parcours
	ELSE	
		bStop := FALSE;	// reprise parcours
	END_IF
	
	//change de tâche si il est bloqué depuis trop longtemps
	IF delay(time_since_enemi_detect,tTimeBeforeAbort) AND bstop THEN 
		bAbort := TRUE;
	ELSE
		bAbort := FALSE;
	END_IF
END_IF;

//______________________________________________________________________________________________________________________________________________
//
// Gestion de la visu 
//______________________________________________________________________________________________________________________________________________
M_visu();

METHOD PUBLIC _M_Angle_enemi : LREAL
VAR_INPUT
	Time_Tour			: LREAL;	// temps du tour
	Time_DetecEnnemi	: LREAL;	//temps de détection d'un ennemi
	Time_FinDetection	: LREAL;	//Temps entre la référence et la fin de la détection d'un ennemi
END_VAR
// Si la balise tourne, l'angle de détection est calculé
IF (Time_Tour > 0) THEN																				//														  Temps:	|	Time_Tour	|	Time_FinDetection - Demi angle
	_M_Angle_enemi := ((360*Time_FinDetection/Time_Tour) - (360*Time_DetecEnnemi)/(Time_Tour*2));	// calcul angle position recepteur avec règle de trois = --------------------------------------------------------------
																									//														  Angle:	|	360° (2*PI)	|		Angle (ce qu'on cherche)
	IF (_M_Angle_enemi < 0) THEN
		_M_Angle_enemi	:= _M_Angle_enemi + 360;// Si le calcul donne une valeur négative, elle est remise en positive
	END_IF																						
END_IF
END_METHOD

METHOD PUBLIC _M_Distance_enemi : LREAL
VAR_INPUT
	Time_Tour			: LREAL;	// temps du tour
	Time_DetecEnnemi	: LREAL;	//temps de détection d'un ennemi
	Time_FinDetection	: LREAL;	//Temps entre la référence et la fin de la détection d'un ennemi
END_VAR
VAR_INST
	Angle_Detection	:	LREAL;		// angle de détection ("largeur" de l'ennemi), toujours en [ns]
END_VAR
// Si la balise tourne, l'angle de détection est calculé
IF (Time_Tour > 0) THEN											//															Temps:	|	Time_Tour	|	Time_DetecEnnemi
	Angle_Detection := (2*PI* Time_DetecEnnemi)/(Time_Tour); 	// calcul angle complet de détection avec règle de trois = ------------------------------------------------
																//															Angle:	|	360° (2PI)	|	Angle_Detection
										
	IF Angle_Detection/2 <> 0 THEN														//											  	 rayon du catadioptre
        _M_Distance_enemi := ABS (uirayonCatadioptre/ TAN(Angle_Detection /2));			//	calcul distance avec trigo :  Distance = -------------------------------
	END_IF																				//											TAN[demi angle détection balise]
END_IF;
END_METHOD

METHOD PUBLIC M_visu 
VAR_INST
	AngleRelativeRAD1 : LREAL;
	AngleRelativeRAD2 : LREAL;
	AngleRelativeRAD3 : LREAL;
END_VAR
IF balise_active AND delay(past_time, T#2S) AND bactivateVisu THEN 

	//adapation des valeurs du 1er récepteur pour les afficher sur la visu
	IF (G_Balise.ArrayEnnemi [0,E_Balise.Angle] < 9000) AND (G_Balise.ArrayEnnemi [0,E_Balise.Distance] < 9000)  THEN;	
		Nothing1 := 0;
		AngleRAD := ((G_Balise.ArrayEnnemi [0,0])*2*PI)/360;
		posiX1 := (SIN (AngleRAD)*(G_Balise.ArrayEnnemi [0,E_Balise.Distance]));
		posiY1 := (COS (AngleRAD)*(G_Balise.ArrayEnnemi [0,E_Balise.Distance]));
		
		AngleRelativeRAD1 := G_Odometrie.lrAngle - AngleRAD;
		
		IF AngleRelativeRAD1 > 2*PI THEN 
			AngleRelativeRAD1 := AngleRelativeRAD1 - 2*PI;
		ELSIF AngleRelativeRAD1 < 0 THEN 
			AngleRelativeRAD1 := AngleRelativeRAD1 + 2*PI;				
		END_IF
		
		coordX1 := G_Odometrie.lrPositionX + (COS(AngleRelativeRAD1) * G_Balise.ArrayEnnemi [0,1]);
		coordY1 := -(G_Odometrie.lrPositionY + (SIN(AngleRelativeRAD1) * G_Balise.ArrayEnnemi [0,1]));
		
		G_Balise.lrCoord_X1 := coordX1;
		G_Balise.lrCoord_Y1 := -coordY1;
		
	ELSIF (G_Balise.ArrayEnnemi [0,E_Balise.Angle] = 9000) AND (G_Balise.ArrayEnnemi [0,E_Balise.Distance] = 9000) AND balise_active THEN ;	
		Nothing1 := 1;
		G_Balise.lrCoord_X1 := -9000;
		G_Balise.lrCoord_X1 := -9000;
	END_IF   
	//adapation des valeurs du 2eme récepteur pour les afficher sur la visu
	IF (G_Balise.ArrayEnnemi [1,E_Balise.Angle] < 9000) AND (G_Balise.ArrayEnnemi [1,E_Balise.Distance] < 9000) THEN;
		Nothing2 := 0;	
		AngleRAD2 := ((G_Balise.ArrayEnnemi [1,0])*2*PI)/360;
		posiX2 := (SIN (AngleRAD2)*(G_Balise.ArrayEnnemi [1,E_Balise.Distance]));
		posiY2 := (COS (AngleRAD2)*(G_Balise.ArrayEnnemi [1,E_Balise.Distance]));
		coordX2 := G_Odometrie.lrPositionX + posiX2;
		coordY2 := G_Odometrie.lrPositionY + posiY2;
		
		AngleRelativeRAD2 := G_Odometrie.lrAngle - AngleRAD2;
		
		IF AngleRelativeRAD2 > 2*PI THEN 
			AngleRelativeRAD2 := AngleRelativeRAD2 - 2*PI;
		ELSIF AngleRelativeRAD2 < 0 THEN 
			AngleRelativeRAD2 := AngleRelativeRAD2 + 2*PI;				
		END_IF
		
		coordX2 := G_Odometrie.lrPositionX + (COS(AngleRelativeRAD2) * G_Balise.ArrayEnnemi [1,E_Balise.Distance]);
		coordY2 := -(G_Odometrie.lrPositionY + (SIN(AngleRelativeRAD2) * G_Balise.ArrayEnnemi [1,E_Balise.Distance]));
		
		G_Balise.lrCoord_X2 := coordX2;
		G_Balise.lrCoord_Y2 := -coordY2;
		
	ELSIF (G_Balise.ArrayEnnemi [0,E_Balise.Angle] = 9000) AND (G_Balise.ArrayEnnemi [0,E_Balise.Distance] = 9000) AND balise_active  THEN;
		Nothing2 := 1;
		G_Balise.lrCoord_X1 := -9000;
		G_Balise.lrCoord_Y1 := -9000;
	END_IF
	//adapation des valeurs du 3eme récepteur pour les afficher sur la visu
	IF (G_Balise.ArrayEnnemi [2,E_Balise.Angle] < 9000) AND (G_Balise.ArrayEnnemi [2,E_Balise.Distance] < 9000) THEN;
		Nothing3 := 0;	
		AngleRAD3 := ((G_Balise.ArrayEnnemi [2,0])*2*PI)/360;
		posiX3 := (SIN (AngleRAD3)*(G_Balise.ArrayEnnemi [2,E_Balise.Distance]));
		posiY3 := (COS (AngleRAD3)*(G_Balise.ArrayEnnemi [2,E_Balise.Distance]));
		coordX3 := G_Odometrie.lrPositionX + posiX3;
		coordY3 := G_Odometrie.lrPositionY + posiY3;
		
		AngleRelativeRAD3 := G_Odometrie.lrAngle - AngleRAD3;
		
		IF AngleRelativeRAD3 > 2*PI THEN 
			AngleRelativeRAD3 := AngleRelativeRAD3 - 2*PI;
		ELSIF AngleRelativeRAD3 < 0 THEN 
			AngleRelativeRAD3 := AngleRelativeRAD3 + 2*PI;				
		END_IF
		
		coordX3 := G_Odometrie.lrPositionX + (COS(AngleRelativeRAD3) * G_Balise.ArrayEnnemi [2,E_Balise.Distance]);
		coordY3 := -(G_Odometrie.lrPositionY + (SIN(AngleRelativeRAD3) * G_Balise.ArrayEnnemi [2,E_Balise.Distance]));
		
		G_Balise.lrCoord_X3 := coordX3;
		G_Balise.lrCoord_Y3 := -coordY3;
		
	ELSIF (G_Balise.ArrayEnnemi [0,E_Balise.Angle] = 9000) AND (G_Balise.ArrayEnnemi [0,E_Balise.Distance] = 9000) AND balise_active   THEN;
		Nothing3 := 1;	
		G_Balise.lrCoord_X3 := -9000;
		G_Balise.lrCoord_Y3 := -9000;
	END_IF
	
	
	//condition distance 550mm 
	IF (G_Balise.ArrayEnnemi [0,E_Balise.Distance] < 550) AND (G_Balise.ArrayEnnemi [0,1]  <>  0)   THEN;
			D1_40cm := 1;
		ELSE 
			D1_40cm := 0;
	END_IF
	IF (G_Balise.ArrayEnnemi [1,E_Balise.Distance] < 550) AND (G_Balise.ArrayEnnemi [1,1]  <>  0)  THEN;
			D2_40cm := 1;
		ELSE 
			D2_40cm := 0;
	END_IF
	IF (G_Balise.ArrayEnnemi [2,E_Balise.Distance] < 550) AND (G_Balise.ArrayEnnemi [2,1]  <>  0) THEN;
			D3_40cm := 1;
		ELSE 
			D3_40cm := 0;
	END_IF
	
	
	//-------------------------------------------------------------------------------------------------------
	
	//condition 4 position devant, derrière, gauche, droite	pour afficher sur la VISU
	IF 		(D1_40cm AND NOT Nothing1 AND ((G_Balise.ArrayEnnemi [0,E_Balise.Angle]  <= 45) OR (G_Balise.ArrayEnnemi [0,E_Balise.Angle] >= 315)))
		OR	(D2_40cm AND NOT Nothing2 AND ((G_Balise.ArrayEnnemi [1,E_Balise.Angle]  <= 45) OR (G_Balise.ArrayEnnemi [1,E_Balise.Angle] >= 315)))
		OR	(D3_40cm AND NOT Nothing3 AND ((G_Balise.ArrayEnnemi [2,E_Balise.Angle]  <= 45) OR (G_Balise.ArrayEnnemi [2,E_Balise.Angle] >= 315))) THEN
			Angle0deg := 0;
		ELSE 
			Angle0deg := 1;
	END_IF
	IF 		(D1_40cm AND NOT Nothing1 AND (G_Balise.ArrayEnnemi [0,E_Balise.Angle] <= 135) AND (G_Balise.ArrayEnnemi [0,E_Balise.Angle] >= 45))
		OR  (D2_40cm AND NOT Nothing2 AND (G_Balise.ArrayEnnemi [1,E_Balise.Angle] <= 135) AND (G_Balise.ArrayEnnemi [1,E_Balise.Angle] >= 45))
		OR  (D3_40cm AND NOT Nothing3 AND (G_Balise.ArrayEnnemi [2,E_Balise.Angle] <= 135) AND (G_Balise.ArrayEnnemi [2,E_Balise.Angle] >= 45)) THEN;
			Angle90deg := 0;
		ELSE 
			Angle90deg := 1;
	END_IF
	IF 		(D1_40cm AND NOT Nothing1 AND (G_Balise.ArrayEnnemi [0,E_Balise.Angle] <= 225) AND (G_Balise.ArrayEnnemi [0,E_Balise.Angle] >= 135))
		OR	(D2_40cm AND NOT Nothing2 AND (G_Balise.ArrayEnnemi [1,E_Balise.Angle] <= 225) AND (G_Balise.ArrayEnnemi [1,E_Balise.Angle] >= 135))
		OR	(D3_40cm AND NOT Nothing3 AND (G_Balise.ArrayEnnemi [2,E_Balise.Angle] <= 225) AND (G_Balise.ArrayEnnemi [2,E_Balise.Angle] >= 135)) THEN;
			Angle180deg := 0;
		ELSE 
			Angle180deg := 1;
	END_IF
	IF 		(D1_40cm AND NOT Nothing1 AND (G_Balise.ArrayEnnemi [0,E_Balise.Angle] <= 315) AND (G_Balise.ArrayEnnemi [0,E_Balise.Angle] >= 225))
		OR	(D2_40cm AND NOT Nothing2 AND (G_Balise.ArrayEnnemi [1,E_Balise.Angle] <= 315) AND (G_Balise.ArrayEnnemi [1,E_Balise.Angle] >= 225))
		OR	(D3_40cm AND NOT Nothing3 AND (G_Balise.ArrayEnnemi [2,E_Balise.Angle] <= 315) AND (G_Balise.ArrayEnnemi [2,E_Balise.Angle] >= 225)) THEN;
			Angle270deg := 0;
		ELSE 
			Angle270deg := 1;
	END_IF
	
	// Chargement des valeurs dans la visualisation
	G_Balise.lrAngle_1		:= G_Balise.ArrayEnnemi [0,E_Balise.Angle];
	G_Balise.lrAngle_2		:= G_Balise.ArrayEnnemi [1,E_Balise.Angle];
	G_Balise.lrAngle_3		:= G_Balise.ArrayEnnemi [2,E_Balise.Angle];
	G_Balise.lrDistance_1	:= G_Balise.ArrayEnnemi [0,E_Balise.Distance];
	G_Balise.lrDistance_2	:= G_Balise.ArrayEnnemi [1,E_Balise.Distance];
	G_Balise.lrDistance_3	:= G_Balise.ArrayEnnemi [2,E_Balise.Distance];
END_IF;
END_METHOD

END_FUNCTION_BLOCK

// ---- POUs/Utillity/Temporisation/delay.TcPOU
FUNCTION delay : bool
VAR_INPUT
	last_time : TIME;
	tempo : TIME;
END_VAR
VAR
END_VAR

IF TIME() - last_time >= tempo THEN 
	delay := TRUE ;
ELSE
	delay := FALSE;
END_IF

END_FUNCTION

// ---- POUs/Interruption/FB_Timeout.TcPOU
FUNCTION_BLOCK FB_Timeout
VAR_INPUT
	match_time 	: TIME;
	max_time	: TIME;
END_VAR
VAR_OUTPUT
	bstop		: BOOL;
END_VAR

//si le temps de match est dépassé, renvoie un signal d'arrêt 
IF match_time >= max_time THEN 
	bstop := TRUE;
ELSE
	bstop := FALSE;
END_IF

END_FUNCTION_BLOCK

// ---- POUs/Motion/ITMotion.TcPOU
PROGRAM ITMotion
VAR
	odometrie 			:FB_Motion_Odometrie;
END_VAR
VAR_INPUT
	IbPower				:BOOL;
	IbStop				:BOOL;
	IbPause				:BOOL;
	IbReset				:BOOL;
END_VAR
VAR_OUTPUT
	QbMoteurOn		:BOOL;
	QbMouvementTermine 	:BOOL;
END_VAR
VAR // added by the converter: edge detectors and wires of the graphical bodies
    _w1, _w2, _w3, _w4 : BOOL;
END_VAR

_w2 := IbPower AND NOT _w1;
_w3 := IbStop OR IbReset;
_w1 := IbStop OR IbReset;
G_Moteurs.mcPowerG(
    Axis := G_Moteurs.axMoteurG,
    Enable := _w2,
    Enable_Positive := true,
    Enable_Negative := true); // MC_Power
G_Moteurs.mcSuperPosD(
    Axis := G_Moteurs.axMoteurD,
    Mode := SUPERPOSITIONMODE_LENGTHREDUCTION_LIMITEDMOTION,
    VelocityDiff := 1600,
    VelocityProcess := 1000,
    Length := 200); // MC_MoveSuperImposed
G_Moteurs.mcSuperPosG(
    Axis := G_Moteurs.axMoteurG,
    Mode := SUPERPOSITIONMODE_LENGTHREDUCTION_LIMITEDMOTION,
    VelocityDiff := 1600,
    VelocityProcess := 1000,
    Length := 200); // MC_MoveSuperImposed
G_Moteurs.mcResetGau(Axis := G_Moteurs.axMoteurG, Execute := IbReset); // MC_Reset
G_Moteurs.mcStopG(Axis := G_Moteurs.axMoteurG, Execute := IbStop, Deceleration := 4000, Jerk := 10000); // MC_Stop
QbMouvementTermine := odometrie.bMouvementDone;
_w4 := IbPower AND NOT _w3;
G_Moteurs.mcRelativeG(Axis := G_Moteurs.axMoteurG, BufferMode := MC_BlendingPrevious); // MC_MoveRelative
odometrie(
    lrPosDepartatelierX := 400,
    lrPosDepartbureauX := 1500,
    lrPosDepartatelierY := 400,
    lrPosDepartbureauY := 730,
    lrAngleDepartatelier := 0,
    lrAngleDepartbureau := PI/2,
    lrEntraxeRoues := 165,
    lrEntraxeRoueFolles := 240); // FB_Motion_Odometrie
G_Moteurs.mcResetDro(Axis := G_Moteurs.axMoteurD, Execute := IbReset); // MC_Reset
G_Moteurs.mcHaltDroite(
    Axis := G_Moteurs.axMoteurD,
    Execute := IbPause,
    Deceleration := 4000,
    Jerk := 10000,
    BufferMode := Tc2_MC2.MC_Aborting); // MC_Halt
G_Moteurs.mcPowerD(
    Axis := G_Moteurs.axMoteurD,
    Enable := _w4,
    Enable_Positive := true,
    Enable_Negative := true); // MC_Power
G_Moteurs.mcStopD(Axis := G_Moteurs.axMoteurD, Execute := IbStop, Deceleration := 4000, Jerk := 10000); // MC_Stop
G_Moteurs.mcRelativeD(Axis := G_Moteurs.axMoteurD, BufferMode := MC_BlendingPrevious); // MC_MoveRelative
G_Moteurs.mcHaltGauche(
    Axis := G_Moteurs.axMoteurG,
    Execute := IbPause,
    Deceleration := 4000,
    Jerk := 10000,
    BufferMode := Tc2_MC2.MC_Aborting); // MC_Halt
QbMoteurOn := odometrie.bMotorPowered;

END_PROGRAM

// ---- POUs/Motion/FB_Motion_Odometrie.TcPOU
FUNCTION_BLOCK FB_Motion_Odometrie
VAR_INPUT
	lrPosDepartatelierX 	:LREAL  ; 	// Position de départ côté atelier en X
	lrPosDepartatelierY 	:LREAL  ; 	// Position de départ côté atelier en Y
	lrAngleDepartatelier	:LREAL  ;	// Angle de départ côté atelier 
	
	lrPosDepartbureauX 		:LREAL  ; 	// Position de départ côté bureau en X
	lrPosDepartbureauY 		:LREAL  ; 	// Position de départ côté bureau en Y
	lrAngleDepartbureau		:LREAL  ;	// Angle de départ côté bureau
	
	lrEntraxeRoues			: LREAL ;	// Entraxe des roues du robot, à mesurer sur le robot
	lrEntraxeRoueFolles		: LREAL	;	// Entraxe des roues folles du robot, à mesurer sur le robot
END_VAR
VAR_OUTPUT
	bMotorPowered			: BOOL;
	bMouvementDone			: BOOL;
END_VAR
VAR //odométrie
 	lrGPosT 				:LREAL; 			//position moteur gauche
	lrDPosT 				:LREAL; 			//position moteur droit
	lrGPosTm1 				:LREAL; 			//position moteur gauche au cycle précédent
	lrDPosTm1 				:LREAL; 			//position moteur droit au cycle précédent
	
	lrGDelta 				:LREAL; 			//Différence de position du moteur gauche entre 2 cycles
	lrDDelta 				:LREAL; 			//Différence de position du moteur droit entre 2 cycles
	lrDelta 				:LREAL; 			//Différence de position au centre du robot entre 2 cycles
	
	lrPositionEncodeurG 	:LREAL; 			// Position de l'encodeur gauche avec facteur lorsqu'on tourne car la roue folle ne tourne pas à la même vitesse que la roue d'entraînement
	lrPositionEncodeurD 	:LREAL; 			// Position de l'encodeur gauche avec facteur lorsqu'on tourne car la roue folle ne tourne pas à la même vitesse que la roue d'entraînement
END_VAR
VAR //pour M_move_curve
	lrCurrentAngle			:LREAL;	
	lrDepartX				:LREAL;
	lrDepartY				:LREAL;
	lrAxeRotationX			:LREAL;
	lrAxeRotationY			:LREAL;
	lrExpectedX 			:LREAL;				//Position finale théorique après une courbe - Alec 08.11.23
	lrExpectedY				:LREAL;				//Position finale théorique après une courbe - Alec 08.11.23
END_VAR

// Axe X est à l'horizontal, l'axe Y est à la verticale, 0-360 degré est dans le sens anti-horaire (sens trigonométrique)

lrGPosT := G_Moteurs.axEncodeurG.NcToPlc.ActPos; // Position Actuelle moteur gauche
lrDPosT := G_Moteurs.axEncodeurD.NcToPlc.ActPos; // Position Actuelle moteur droit

lrGDelta := lrGPosT - lrGPosTm1; // Différence de position du moteur gauche entre les cycles
lrDDelta := lrDPosT - lrDPosTm1; // Différence de position du moteur droit entre les cycles

lrDelta := (1.0/2.0)*(lrGDelta+lrDDelta); // Différence de distance au centre du robot

// Calcul de l'angle :
G_Odometrie.lrAngle := G_Odometrie.lrAngle + ((lrDDelta-lrGDelta) / lrEntraxeRoueFolles); // Angle = périmètre / diamètre

IF G_Odometrie.lrAngle > (2*PI) THEN // Position absolue sur un tour pour l'angle
	G_Odometrie.lrAngle := G_Odometrie.lrAngle - (2*PI); // Si on a tourné plus de 1 tour, on soustrait 360 degrés
END_IF
IF G_Odometrie.lrAngle < 0.0 THEN // Position absolue sur un tour pour l'angle
	G_Odometrie.lrAngle := G_Odometrie.lrAngle + (2*PI); // Si on a tourné plus de 1 tour en négatif, on additionne 360 degrés
END_IF

G_Odometrie.lrPositionX := G_Odometrie.lrPositionX + (lrDelta * COS(G_Odometrie.lrAngle)); //Calcul de la position en X lorsqu'il se déplace en diagonal
G_Odometrie.lrPositionY := G_Odometrie.lrPositionY + (lrDelta * SIN(G_Odometrie.lrAngle)); //Calcul de la position en Y lorsqu'il se déplace en diagonal

lrGPosTm1 := lrGPosT; //Nouvelle position gauche sauvegardée pour le prochain cycle
lrDPosTm1 := lrDPosT; //Nouvelle position droit sauvegardée pour le prochain cycle
																//								360° (tour complet en deg)	 Angle en deg
G_Odometrie.lrAngleDeg := G_Odometrie.lrAngle * 360 / (2*PI);   // Valeur de l'angle en degré : -------------------------- = ------------- (on peut simplifier par 2 le 360 et le 2*PI)
																//								2*PI (tour complet en rad)	 Angle en rad										
//OUTPUT
bMouvementDone := G_Moteurs.mcRelativeG.Done AND G_Moteurs.mcRelativeD.Done;
bMotorPowered := G_Moteurs.mcPowerG.Busy and G_Moteurs.mcPowerD.Busy;

METHOD PRIVATE _M_ATAN2 : LREAL
VAR_INPUT
	X : LREAL; //côté opposé
	Y : LREAL; //côté adjacent
END_VAR
VAR
END_VAR
IF X > 0.0 THEN			
		_M_ATAN2 := ATAN(Y/X);		// Quand X est plus grand que 0, on divise Y par X
ELSIF X < 0.0 THEN
	IF Y >=0.0 THEN
		_M_ATAN2 := ATAN(Y/X) + PI;	// Quand X est plus petit que 0, mais pas Y, on ajoute PI (180°) à l'angle calculé
	ELSE
		_M_ATAN2 := ATAN(Y/X) - PI;	// Quand X et Y sont plus petits que 0, on enlève PI (180°) à l'angle calculé
	END_IF;
	
ELSIF Y > 0.0 THEN
	_M_ATAN2 := PI*0.5;				// Si X est à 0 et Y est plus grand que 0, l'angle est de PI/2 (90°)
ELSIF Y < 0.0 THEN
    _M_ATAN2 := -PI*0.5;			// Si X est de 0 et Y est plus petit que 0, l'angle est de -PI/2 (-90°)
ELSE
   _M_ATAN2 := 0.0;					// Quand X et Y sont égals à 0, l'angle est de 0
END_IF;
END_METHOD

METHOD PRIVATE _M_coord2angle : LREAL
VAR_INPUT
	x 				:LREAL;	//position du robot voulu sur l'axe X
	y 				:LREAL;	//position voulu du robot sur l'axe Y
	bbackward		:BOOL := FALSE;  //déplacement avec l'arrière du robot 
END_VAR
VAR
	lrangle_to_move :LREAL; // angle dont le robot va devoir tourner
	lrmove_a 		:LREAL;
END_VAR
// Calcul de l'angle à parcourir avec de la trigonometrie (arctan(op/adj) = angle)
lrangle_to_move := G_Odometrie.lrAngle - _M_ATAN2(		// La fonction ATAN2 sert à faire arctan en évitant les divisions par 0
X := (x - G_Odometrie.lrPositionX), 
Y := (y - G_Odometrie.lrPositionY)); //x,y pour atan2, le calcul est fait en radians
	
//si le robot dois aller en marche arrière la rotation est incrémentée de PI (180°) pour qu'elle soit juste 
IF bbackward AND lrangle_to_move - PI < 0  THEN
		lrangle_to_move := lrangle_to_move + PI;
ELSIF bbackward AND lrangle_to_move - PI >= 0  THEN
		lrangle_to_move := lrangle_to_move - PI;
END_IF

// Si l'angle à parcourir est plus petit que 0° ou plus grand que 2PI(360°), on lui ajoute/enlève 360° pour qu'il ne le soit plus
IF lrangle_to_move < 0 THEN
	lrangle_to_move := 2*PI + lrangle_to_move;
ELSIF lrangle_to_move > 2*PI THEN
	lrangle_to_move := lrangle_to_move - 2*PI;
END_IF

// Les distance que les roues doivenet parcourir pour faire la rotation demandée, sont envoyées au MC_MoveRelative
IF lrangle_to_move = 0 THEN
		lrmove_a := 0;
		G_Moteurs.mcRelativeD.Distance := lrmove_a;
		G_Moteurs.mcRelativeG.Distance := - lrmove_a;
ELSIF lrangle_to_move < PI THEN		// On tourne dans le sens horaire 		//																		Angle [rad]						Angle[°]
		lrmove_a := lrEntraxeRoues * (ABS(lrangle_to_move/2));	// Calclul de la distance avec le rayon et l'angle|Distance = Rayon* -----------------  (PI* Rayon*  ---------)
		G_Moteurs.mcRelativeD.Distance := - lrmove_a;						//																			2							360
		G_Moteurs.mcRelativeG.Distance :=   lrmove_a;
ELSIF lrangle_to_move >= PI THEN		// On tourne dans le sens anti-horaire
		lrmove_a := lrEntraxeRoues * (ABS((2*PI-lrangle_to_move)/2));
		G_Moteurs.mcRelativeD.Distance :=   lrmove_a;
		G_Moteurs.mcRelativeG.Distance := - lrmove_a;
		
END_IF
_M_coord2angle := lrangle_to_move;
END_METHOD

METHOD PRIVATE _M_coord2distance : LREAL
VAR_INPUT
	x 				:LREAL;
	y 				:LREAL; 
	bbackward		:BOOL := FALSE;  //déplacement avec l'arrière du robot 
END_VAR
VAR
	lrdelta_distance 	:LREAL;
END_VAR
// Calcul de la distance à parcourir par pythagore (Racine carrée de (x au carré plus y au carré))
lrdelta_distance := SQRT(		// SQRT = racine carrée
	EXPT(ABS(x - G_Odometrie.lrPositionX),2) + EXPT(ABS(y - G_Odometrie.lrPositionY),2)); // EXPT = exponantielle (puissance), ABS = valeur absolue
	
//inversion de la valeur de distance du robot pour le faire rouler en marche arrière
IF bbackward THEN
	lrdelta_distance := -lrdelta_distance;
END_IF

// La distance à parcourir calculée, est envoyée aux MC_MoveRelative
G_Moteurs.mcRelativeD.Distance := lrdelta_distance;
G_Moteurs.mcRelativeG.Distance := lrdelta_distance;
_M_coord2distance := lrdelta_distance;
END_METHOD

METHOD PUBLIC M_init_coordonne : BOOL
VAR_INPUT
	bChoixCote : BOOL; //True = atelier, FALSE = bureau
END_VAR
VAR_OUTPUT
	bDone : bool;
END_VAR
IF bChoixCote THEN 	
	G_Odometrie.lrAngle := lrAngleDepartAtelier ; //(5*PI)/4;  
	G_Odometrie.lrPositionX := lrPosDepartAtelierX;
	G_Odometrie.lrPositionY := lrPosDepartAtelierY;
ELSE								
	G_Odometrie.lrAngle := lrAngleDepartBureau; //(3*PI)/4; //Le robot est décalé de 180 degré pour avoir l'avant dans le sens de la table
	G_Odometrie.lrPositionX := lrPosDepartBureauX ;
	G_Odometrie.lrPositionY := lrPosDepartBureauY ;
END_IF
bDone := True;
END_METHOD

METHOD PUBLIC M_move_curve : BOOL
VAR_INPUT
	lrRayon				:LREAL;	//positif => droite, negatif => gauche
	lrAngle				:LREAL;	//positif => marche avant, negatif => marche arrière
	lrSpeed				:LREAL;	// vitesse voulue du robot
	bExecute			:BOOL;	//execution du function bloc
END_VAR
VAR_OUTPUT
	bDone 				:BOOL;
END_VAR

VAR_INST
	lrArcX 				:LREAL;
	lrArcY				:LREAL;
	lrVecteurDepart		:ARRAY [0..1] OF LREAL; //vecteur entre l'axe de rotation et le point de départ du robot
	lrVecteurPosition	:ARRAY [0..1] OF LREAL; //vecteur entre l'axe de rotation et la position actuelle du robot
	lrVecteurTrajectoire:ARRAY [0..1] OF LREAL; //vecteur de la positon théorique du robot en fonction de l'ange auxquel il se trouve
	
	lrProduitVecteur	:LREAL;
	lrSommeNormeVecteur	:LREAL;
	lrDifferencePosition:LREAL;

	
	step 				:USINT; 
	r_trig 				:R_TRIG;
	lrCorrectionValue 	:LREAL := 0.1;	
	bBackward 			:BOOL;
END_VAR
//Prototype, à tester avant d'utiliser


r_trig(CLK := bExecute);
bdone := FALSE;
CASE step OF 
	0:
		IF r_trig.Q THEN
			lrCurrentAngle := 0;
			lrDepartX := G_Odometrie.lrPositionX;
			lrDepartY := G_Odometrie.lrPositionY;
			lrAxeRotationX := G_Odometrie.lrPositionX + lrRayon*COS(G_Odometrie.lrAngle - PI/2);
			lrAxeRotationY := G_Odometrie.lrPositionY + lrRayon*SIN(G_Odometrie.lrAngle - PI/2);
			lrVecteurDepart[0] := lrDepartX-lrAxeRotationX;
			lrVecteurDepart[1] := lrDepartY-lrAxeRotationY;
			step := step + 1;
		END_IF
	1:
		IF NOT G_Moteurs.mcRelativeD.Execute AND NOT G_Moteurs.mcRelativeG.Execute THEN
			//En Avant
			IF lrAngle > 0 THEN
				bBackward := FALSE;
				IF lrRayon > 0 THEN 	//rotation vers la droite
					G_Moteurs.mcRelativeD.Distance := DEGRE2RAD(lrAngle-lrCurrentAngle)*(lrRayon - lrEntraxeRoues/2);
					G_Moteurs.mcRelativeG.Distance := DEGRE2RAD(lrAngle-lrCurrentAngle)*(lrRayon + lrEntraxeRoues/2);
					G_Moteurs.mcRelativeD.velocity := (G_Moteurs.mcRelativeD.Distance/G_Moteurs.mcRelativeG.Distance) * lrspeed;	//si coodronnées attribuées aux moteurs, exécution du mouvement prévu
					G_Moteurs.mcRelativeG.Velocity := lrspeed;	//si coodronnées attribuées aux moteurs, exécution du mouvement prévu
					lrAngle := DEGRE2RAD(lrAngle);
					lrExpectedX := lrAxeRotationX + lrVecteurDepart[0]*COS(lrAngle) + lrVecteurDepart[1]*SIN(lrAngle);
					lrExpectedY := lrAxeRotationY -lrVecteurDepart[0]*SIN(lrAngle) + lrVecteurDepart[1]*COS(lrAngle);
				ELSIF lrRayon < 0 THEN 	// rotation vers la gauche
					lrArcX := lrRayon*(COS(DEGRE2RAD(lrAngle-lrCurrentAngle) - 1));
					lrArcY := lrRayon*SIN(DEGRE2RAD(lrAngle-lrCurrentAngle));
					//matrice rotation
					lrExpectedX := lrArcX * COS(G_Odometrie.lrAngle - PI/2) - lrArcY * SIN(G_Odometrie.lrAngle - PI/2);
					lrExpectedY := lrArcX * SIN(G_Odometrie.lrAngle - PI/2) + lrArcY * COS(G_Odometrie.lrAngle - PI/2);
					lrExpectedX := G_Odometrie.lrPositionX + lrExpectedX;
					lrExpectedY := G_Odometrie.lrPositionY + lrExpectedY;
						
					lrRayon := ABS(lrRayon);
					G_Moteurs.mcRelativeD.Distance := DEGRE2RAD(lrAngle-lrCurrentAngle)*(lrRayon + lrEntraxeRoues/2);
					G_Moteurs.mcRelativeG.Distance := DEGRE2RAD(lrAngle-lrCurrentAngle)*(lrRayon - lrEntraxeRoues/2);
					G_Moteurs.mcRelativeG.Acceleration := (G_Moteurs.mcRelativeD.Distance/G_Moteurs.mcRelativeG.Distance)*2000;
					G_Moteurs.mcRelativeD.Acceleration := 2000;
					G_Moteurs.mcRelativeD.Deceleration := G_Moteurs.mcRelativeD.Acceleration;
					G_Moteurs.mcRelativeG.Deceleration := G_Moteurs.mcRelativeG.Acceleration;
					G_Moteurs.mcRelativeD.Velocity := lrspeed;	//si coodronnées attribuées aux moteurs, exécution du mouvement prévu
					G_Moteurs.mcRelativeG.velocity := (G_Moteurs.mcRelativeG.Distance/G_Moteurs.mcRelativeD.Distance) * lrspeed;	//si coodronnées attribuées aux moteurs, exécution du mouvement prévu
				END_IF	
			//En Arrière	
			ELSIF lrAngle < 0 THEN
				bBackward := TRUE;
				lrAngle := ABS(lrAngle);
				IF lrRayon > 0 THEN 	//rotation vers la droite
					G_Moteurs.mcRelativeD.Distance := -(DEGRE2RAD(lrAngle-lrCurrentAngle)*(lrRayon - lrEntraxeRoues/2));
					G_Moteurs.mcRelativeG.Distance := -(DEGRE2RAD(lrAngle-lrCurrentAngle)*(lrRayon + lrEntraxeRoues/2));
					G_Moteurs.mcRelativeD.Acceleration := (G_Moteurs.mcRelativeD.Distance/G_Moteurs.mcRelativeG.Distance)*2000;
					G_Moteurs.mcRelativeG.Acceleration := 2000;
					G_Moteurs.mcRelativeD.Deceleration := G_Moteurs.mcRelativeD.Acceleration;
					G_Moteurs.mcRelativeG.Deceleration := G_Moteurs.mcRelativeG.Acceleration;
					G_Moteurs.mcRelativeD.velocity := (G_Moteurs.mcRelativeD.Distance/G_Moteurs.mcRelativeG.Distance) * lrspeed;	//si coodronnées attribuées aux moteurs, exécution du mouvement prévu
					G_Moteurs.mcRelativeG.Velocity := lrspeed;	//si coodronnées attribuées aux moteurs, exécution du mouvement prévu
					
				ELSIF lrRayon < 0 THEN 	// rotation vers la gauche
					lrRayon := ABS(lrRayon);
					G_Moteurs.mcRelativeD.Distance := -(DEGRE2RAD(lrAngle-lrCurrentAngle)*(lrRayon + lrEntraxeRoues/2));
					G_Moteurs.mcRelativeG.Distance := -(DEGRE2RAD(lrAngle-lrCurrentAngle)*(lrRayon - lrEntraxeRoues/2));
					G_Moteurs.mcRelativeG.Acceleration := (G_Moteurs.mcRelativeD.Distance/G_Moteurs.mcRelativeG.Distance)*2000;
					G_Moteurs.mcRelativeD.Acceleration := 2000;
					G_Moteurs.mcRelativeD.Deceleration := G_Moteurs.mcRelativeD.Acceleration;
					G_Moteurs.mcRelativeG.Deceleration := G_Moteurs.mcRelativeG.Acceleration;
					G_Moteurs.mcRelativeD.Velocity := lrSpeed;	//si coodronnées attribuées aux moteurs, exécution du mouvement prévu
					G_Moteurs.mcRelativeG.velocity := (G_Moteurs.mcRelativeG.Distance/G_Moteurs.mcRelativeD.Distance) * lrspeed;	//si coodronnées attribuées aux moteurs, exécution du mouvement prévu
				END_IF
			END_IF
	 	END_IF;
		
		G_Moteurs.mcRelativeD.Execute := TRUE;	//si coodronnées attribuées aux moteurs, exécution du mouvement prévu
		G_Moteurs.mcRelativeG.Execute := TRUE;	//si coodronnées attribuées aux moteurs, exécution du mouvement prévu
		
		//position en temps réel 
		IF NOT bBackward THEN 	//marche avant
			IF lrRayon > 0 THEN //rotation vers la droite
				//angle entre 2 vecteurs => théorème du produit de vecteur
				lrVecteurPosition[0] := G_Odometrie.lrPositionX-lrAxeRotationX;
				lrVecteurPosition[1] := G_Odometrie.lrPositionY-lrAxeRotationY;
				
				lrProduitVecteur := (lrVecteurPosition[0]*lrVecteurDepart[0])+(lrVecteurPosition[1]*lrVecteurDepart[1]);
				lrSommeNormeVecteur := HYP(lrVecteurDepart[0],lrVecteurDepart[1]) * HYP(lrVecteurPosition[0],lrVecteurPosition[1])+1E-100;
				lrCurrentAngle := ACOS(lrProduitVecteur/lrSommeNormeVecteur);
								
				lrVecteurTrajectoire[0] := lrAxeRotationX + lrVecteurDepart[0]*COS(lrCurrentAngle) + lrVecteurDepart[1]*SIN(lrCurrentAngle);
				lrVecteurTrajectoire[1] := lrAxeRotationY - lrVecteurDepart[0]*SIN(lrCurrentAngle) + lrVecteurDepart[1]*COS(lrCurrentAngle);
				lrDifferencePosition := HYP(lrVecteurTrajectoire[0]-G_Odometrie.lrPositionX,lrVecteurTrajectoire[1]-G_Odometrie.lrPositionY);

				IF lrDifferencePosition > 5 AND NOT PlusOuMoins(lrCurrentAngle,lrAngle,PI/36)THEN
					G_Moteurs.mcSuperPosG.Distance :=  lrCorrectionValue * lrDifferencePosition;
					G_Moteurs.mcSuperPosD.Distance :=  0;
					G_Moteurs.mcSuperPosG.Execute := TRUE;
					G_Moteurs.mcSuperPosD.Execute := TRUE; 
				END_IF
				
			ELSIF lrRayon < 0 THEN //rotation vers la gauche
				pass();
			END_IF
		ELSE					//marche arrière 
			IF lrRayon > 0 THEN //rotation vers la droite
				pass();
			ELSIF lrRayon < 0 THEN  // rotation vers la gauche
				pass();
			END_IF
		END_IF
		
		IF G_Moteurs.mcSuperPosD.Done AND G_Moteurs.mcSuperPosG.Done THEN
			G_Moteurs.mcSuperPosG.Execute := FALSE;
			G_Moteurs.mcSuperPosD.Execute := FALSE; 
		END_IF
		
		IF bMouvementDone THEN 
			G_Moteurs.mcRelativeD.Execute := FALSE;	//si coodronnées attribuées aux moteurs, exécution du mouvement prévu
			G_Moteurs.mcRelativeG.Execute := FALSE;	//si coodronnées attribuées aux moteurs, exécution du mouvement prévu
			G_Moteurs.mcSuperPosG.Execute := FALSE;
			G_Moteurs.mcSuperPosD.Execute := FALSE; 
			G_Moteurs.mcRelativeD.distance := 0;	//si coodronnées attribuées aux moteurs, exécution du mouvement prévu
			G_Moteurs.mcRelativeG.distance := 0;	//si coodronnées attribuées aux moteurs, exécution du mouvement prévu
			G_Moteurs.mcRelativeG.Acceleration := 0;
			G_Moteurs.mcRelativeD.Acceleration := 0;
			G_Moteurs.mcRelativeD.Deceleration := 0;
			G_Moteurs.mcRelativeG.Deceleration := 0;
			step := 0;
			bdone := TRUE;
		END_IF
END_CASE
END_METHOD

METHOD PUBLIC M_move_distance : BOOL
VAR_INPUT 
	lrDistance			:LREAL;	// angle désiré du robot en sens anti horaire (cercle trigo)
	lrSpeed				:LREAL;	// vitesse voulue du robot
	bExecute			:BOOL;	//execution du function bloc
END_VAR
VAR_OUTPUT
	bDone 				:BOOL;
END_VAR
VAR_INST
	step 				:USINT; 
	r_trig 				: R_TRIG;
END_VAR
r_trig(CLK := bExecute);
bDone := FALSE;
CASE step OF 
	0:
		IF r_trig.Q THEN
			G_Moteurs.mcRelativeD.velocity := lrspeed;	//si coodronnées attribuées aux moteurs, exécution du mouvement prévu
			G_Moteurs.mcRelativeG.Velocity := lrspeed;	//si coodronnées attribuées aux moteurs, exécution du mouvement prévu
			step := step + 1;
		END_IF
	1:
		G_Moteurs.mcRelativeD.Distance := lrDistance;
		G_Moteurs.mcRelativeG.Distance := lrDistance;
		step := step + 1;
	2:
		G_Moteurs.mcRelativeD.Execute := TRUE;	//si coodronnées attribuées aux moteurs, exécution du mouvement prévu
		G_Moteurs.mcRelativeG.Execute := TRUE;	//si coodronnées attribuées aux moteurs, exécution du mouvement prévu
		IF bMouvementDone THEN 
			G_Moteurs.mcRelativeD.Execute := FALSE;	//si coodronnées attribuées aux moteurs, exécution du mouvement prévu
			G_Moteurs.mcRelativeG.Execute := FALSE;	//si coodronnées attribuées aux moteurs, exécution du mouvement prévu
			G_Moteurs.mcRelativeD.distance := 0;	//si coodronnées attribuées aux moteurs, exécution du mouvement prévu
			G_Moteurs.mcRelativeG.distance := 0;	//si coodronnées attribuées aux moteurs, exécution du mouvement prévu
			bDone := TRUE;
			step := 0;
		END_IF
END_CASE
END_METHOD

METHOD PUBLIC M_move_rotation : BOOL
VAR_INPUT
	lrAngle				:LREAL;	// angle désiré du robot en sens anti horaire (cercle trigo)
	lrSpeed				:LREAL;	// vitesse voulue du robot
	bExecute			:BOOL;	//execution du function bloc
END_VAR
VAR_OUTPUT
	bDone 				:BOOL;
END_VAR
VAR_INST
	step 				:USINT; 
	r_trig 				: R_TRIG;
	lrangle_to_move		:LREAL;	// angle dont le robot va devoir tourner
END_VAR
// fonctionne en faisant plusieurs tours
	// - premier tour:		Counter = 0		mise à 0 des distances à effectuer par les moteurs
	// - deuxième tour:		Counter = 1		Mise en mouvement des moteurs pour la rotation
	// - troisième tour:	Counter = 2		remise à 0 du FB et renvoi d'un "done"

r_trig(CLK := bExecute);
bdone := FALSE;
CASE step OF 
	0:
		IF r_trig.Q THEN
			G_Moteurs.mcRelativeD.velocity := lrspeed;	//si coodronnées attribuées aux moteurs, exécution du mouvement prévu
			G_Moteurs.mcRelativeG.Velocity := lrspeed;	//si coodronnées attribuées aux moteurs, exécution du mouvement prévu
			step := step + 1;
		END_IF
	1:
		lrangle_to_move := lrAngle - G_Odometrie.lrAngleDeg; // définition de l'angle à parcourir
		IF PlusOuMoins(lrangle_to_move, 0.0, 0.2) THEN 
			G_Moteurs.mcRelativeD.Distance := 0;
			G_Moteurs.mcRelativeG.Distance := 0;
		ELSIF lrAngle_to_move < 0 THEN
			lrangle_to_move := ABS(lrangle_to_move);
			IF lrangle_to_move <= 180 THEN
				lrangle_to_move := DEGRE2RAD(lrangle_to_move);
				G_Moteurs.mcRelativeD.Distance := -lrangle_to_move * lrEntraxeRoues / 2;
				G_Moteurs.mcRelativeG.Distance := lrangle_to_move * lrEntraxeRoues / 2;
			ELSIF lrangle_to_move > 180 THEN	//si l'angle est inférieur ou égal à 180, on tourne en sens anti-horaire						Angle[°]
				lrangle_to_move := DEGRE2RAD(lrangle_to_move);
				G_Moteurs.mcRelativeD.Distance := (2*PI - lrangle_to_move) * lrEntraxeRoues / 2;												//							  360
				G_Moteurs.mcRelativeG.Distance := -(2*PI - lrangle_to_move) * lrEntraxeRoues / 2;
			END_IF
		ELSIF lrAngle_to_move > 0 THEN 
			IF lrangle_to_move <= 180 THEN
				lrangle_to_move := DEGRE2RAD(lrangle_to_move);
				G_Moteurs.mcRelativeD.Distance := lrangle_to_move * lrEntraxeRoues / 2;
				G_Moteurs.mcRelativeG.Distance := -lrangle_to_move * lrEntraxeRoues / 2;
			ELSIF lrangle_to_move > 180 THEN	//si l'angle est inférieur ou égal à 180, on tourne en sens anti-horaire						Angle[°]
				lrangle_to_move := DEGRE2RAD(lrangle_to_move);
				G_Moteurs.mcRelativeD.Distance := -(2*PI - lrangle_to_move) * lrEntraxeRoues / 2;												//							  360
				G_Moteurs.mcRelativeG.Distance := (2*PI - lrangle_to_move) * lrEntraxeRoues / 2;
			END_IF	
		END_IF
		step := step + 1; 
	2:
		G_Moteurs.mcRelativeD.Execute := TRUE;	//si coodronnées attribuées aux moteurs, exécution du mouvement prévu
		G_Moteurs.mcRelativeG.Execute := TRUE;	//si coodronnées attribuées aux moteurs, exécution du mouvement prévu
		IF bMouvementDone THEN 
			G_Moteurs.mcRelativeD.Execute := FALSE;	//si coodronnées attribuées aux moteurs, exécution du mouvement prévu
			G_Moteurs.mcRelativeG.Execute := FALSE;	//si coodronnées attribuées aux moteurs, exécution du mouvement prévu
			G_Moteurs.mcRelativeD.distance := 0;	//si coodronnées attribuées aux moteurs, exécution du mouvement prévu
			G_Moteurs.mcRelativeG.distance := 0;	//si coodronnées attribuées aux moteurs, exécution du mouvement prévu
			bdone := TRUE;
			step := 0;
		END_IF
END_CASE
END_METHOD

METHOD PUBLIC M_move_to_coordonne : BOOL
VAR_INPUT	
	x  					:LREAL; //position voulue du robot en X
	y  					:LREAL; //position voulue du robot en Y
	lrspeed 			:LREAL; //vitesse voulue du robot depuis parcours
	bExecute 			:BOOL; 	//permet l'activation du function bloc
	bbackward			:BOOL := FALSE;  //déplacement avec l'arrière du robot 
END_VAR
VAR_OUTPUT
	bDone 				:BOOL;
END_VAR
VAR_INST
	step 				:USINT;	
	r_trig 				:R_TRIG;		//front montant pour marquer la fin d'un déplacement
END_VAR
// fonctionne en faisant plusieurs tours
	// - premier tour:		Counter = 0		mise à 0 des distances à effectuer par les moteurs
	// - deuxième tour:		Counter = 1		rotation pour se tourner vers les coordonnées cibles (si nécessaire uniquement)
	// - troisième tour:	Counter = 2		Déplacement vers les les coordonnées cibles
	// - quatrième tour: 	Counter = 3		remise à 0 du FB et renvoi d'un "done"

// Quand le bloc est activé, le robot fait une rotation puis un déplacement en fonction de sa position actuelle et de la position à atteindre	
r_trig(clk := bexecute);
bdone :=FALSE;
CASE step OF
	0:	//lance l'execution de la fonction
		IF r_trig.q THEN 
			step := step + 1;
			// Réglage de la vitesse de rotation des moteurs
			G_Moteurs.mcRelativeD.Velocity 	:= lrspeed;
			G_Moteurs.mcRelativeG.Velocity	:= lrspeed;
			G_Moteurs.mcRelativeG.Distance 	:= 0;
			G_Moteurs.mcRelativeD.Distance 	:= 0;
		END_IF
	1:
		// attribue les valeurs aux moteurs pour une éventuelle rotation

		_M_coord2angle(x,y,bbackward);		
	
		// S'il n'y a aucune rotation à faire avant de faire un mouvement, le compteur est incrémenté
		IF G_Moteurs.mcRelativeD.Distance = 0 AND G_Moteurs.mcRelativeG.Distance = 0 THEN
			step := step + 1;
		ELSE //Exécution des mouvements relatifs
			G_Moteurs.mcRelativeD.Execute := TRUE;	//si coodronnées attribuées aux moteurs, exécution du mouvement prévu
			G_Moteurs.mcRelativeG.Execute := TRUE;	//si coodronnées attribuées aux moteurs, exécution du mouvement prévu	
			
			IF bMouvementDone THEN
				G_Moteurs.mcRelativeD.Execute := FALSE;	//si pas de coodronnées attribuées aux moteurs, pas d'exécution du mouvement prévu
				G_Moteurs.mcRelativeG.Execute := FALSE;	//si pas de coodronnées attribuées aux moteurs, pas d'exécution du mouvement prévu
				G_Moteurs.mcRelativeG.Distance := 0;
				G_Moteurs.mcRelativeD.Distance := 0;
				step := step + 1;
			END_IF;
		END_IF
	2:
		// atribue les valeurs aux moteurs pour le déplacement
		_M_coord2distance(x,y,bbackward);		
		// S'il n'y a aucun déplacement à faire avant de faire un mouvement, le compteur est incrémenté
		IF G_Moteurs.mcRelativeD.Distance = 0 AND G_Moteurs.mcRelativeG.Distance = 0 THEN
			bdone := TRUE;
			step := 0;
		ELSE //Exécution des mouvements relatifs
			G_Moteurs.mcRelativeD.Execute := TRUE;	//si coodronnées attribuées aux moteurs, exécution du mouvement prévu
			G_Moteurs.mcRelativeG.Execute := TRUE;	//si coodronnées attribuées aux moteurs, exécution du mouvement prévu	
			
			IF bMouvementDone THEN
			G_Moteurs.mcRelativeD.Execute := FALSE;	//si pas de coodronnées attribuées aux moteurs, pas d'exécution du mouvement prévu
			G_Moteurs.mcRelativeG.Execute := FALSE;	//si pas de coodronnées attribuées aux moteurs, pas d'exécution du mouvement prévu
			G_Moteurs.mcRelativeG.Distance := 0;
			G_Moteurs.mcRelativeD.Distance := 0;
			bdone := TRUE;
			step := 0;
			END_IF;
		END_IF
END_CASE
END_METHOD

METHOD PUBLIC M_reset_moteurs : BOOL
VAR_INPUT
END_VAR
G_Moteurs.mcRelativeD.Execute := FALSE;
G_Moteurs.mcRelativeG.Execute := FALSE;
END_METHOD

METHOD PUBLIC M_set_acceleration : BOOL
VAR_INPUT
	lrAcc 	: LREAL;
	lrDecc 	: LREAL;
END_VAR
G_Moteurs.mcRelativeD.Acceleration	:= lrAcc;
G_Moteurs.mcRelativeG.Acceleration	:= lrAcc;
G_Moteurs.mcRelativeD.Deceleration	:= lrDecc;
G_Moteurs.mcRelativeG.Deceleration	:= lrDecc;
END_METHOD

END_FUNCTION_BLOCK

// ---- POUs/Utillity/Maths/DEGRE2RAD.TcPOU
FUNCTION DEGRE2RAD : lreal
VAR_INPUT
	lrAngle : LREAL;
END_VAR
VAR
END_VAR

DEGRE2RAD := lrAngle*PI/180;

END_FUNCTION

// ---- POUs/Utillity/Maths/HYP.TcPOU
FUNCTION HYP : lreal
VAR_INPUT
	X :LREAL;
	Y :LREAL;
END_VAR
VAR
END_VAR

HYP := sqrt(expt(X,2)+expt(Y,2));

END_FUNCTION

// ---- POUs/Utillity/Logic/plusOuMoins.TcPOU
FUNCTION plusOuMoins : bool
VAR_INPUT
	val1  : LREAL;
	val2  : LREAL;
	plage : LREAL;
END_VAR

IF val1 < val2 + plage AND val1 > val2 - plage THEN 
	plusOuMoins := TRUE;
ELSE
	plusOuMoins := FALSE;
END_IF

END_FUNCTION

// ---- POUs/MAIN.TcPOU
PROGRAM MAIN
VAR
	EtapeEnCours:string(50);
END_VAR
VAR // added by the converter: edge detectors and wires of the graphical bodies
    _w1, _w3, _w4, _w5, _w6, _w7, _w8, _w10 : ANY;
    _w2, _w9 : BOOL;
END_VAR

// note: this text did not pass the execution check against the stored diagram
// Bobst Robot Team
// Visual Components Framework
// Alec Horth17.01.2024
// Structure_MAIN
// Contrôle les autres composants et la machine d'état du robot
//
// ITAction
// Gère les fonctions spécifiques aux actions du robot. Il doit être adapté
// selon les besoins entre chaque années
EtapeEnCours := _w1;
_w3 := _w2 OR G_Visus.bInitStartPyscript;
ITInterruption(IbStartBalise := _w4, IbMatchEnCours := _w5, IbStartVisuBalise := true, IbRestartTwincat := G_Visus.bMenuRestart, IbArretDetection := G_Match.Tableau[G_Match.iLigne].bArretDetection);
G_Visus.bInitPyScriptRunning := _w6;
ITMotion(IbPower := _w7, IbStop := _w8, IbPause := ITInterruption.QbPauseMotion, IbReset := ITInterruption.QbResetMotion);
_w8 := _w9 OR ITInterruption.QbStopMotion;
ITCommunication_0(); // ITCommunication
Structure_MAIN(IbStartInit := G_Visus.bInitStart, IbStartMatch := G_IO.bCaptDepart or G_Visus.bInitStartMatch, IbChoixCote := G_Visus.bInitChoixCote, IiChoixParcours := G_Visus.iInitChoixParcours, IbMoteurOn := ITMotion.QbMoteurOn, IbPauseMotion := ITInterruption.QbPauseMotion, IbEndMatch := ITInterruption.QbEndMatch, IbAbortTask := ITInterruption.QbAbortTask, IbPyScriptActive := _w6, IiNumDynamixel := _w10);
ITAction(IbStartPyscript := _w3, IbStopPyscript := G_Visus.bInitStopPyscript);

END_PROGRAM

// ---- POUs/Structure/Structure_MAIN.TcPOU
PROGRAM Structure_MAIN
VAR
	baseTime:TIME; //tempo universel à utiliser n'importe où avec la fonction delay()
	tempTableau:ST_Tableau;
END_VAR
VAR_INPUT
	IbStartInit: BOOL;
	IbStartMatch: BOOL;
	IbChoixCote: BOOL;
	IiChoixParcours: INT;
	IbMoteurOn:BOOL;
	IbPauseMotion : BOOL;
	IbEndMatch:BOOL;
	IbAbortTask:BOOL;
	IbPyScriptActive : BOOL;
	IiNumDynamixel:INT;
END_VAR
VAR_OUTPUT
	QbmoteurPower:BOOL;
	QbmoteurStop:BOOL;
	QbstartBalise:BOOL;
	QbMatchEnCours:BOOL;
	QbstartPyScript:BOOL;
	QbEtapeEnCours:STRING(50);
END_VAR

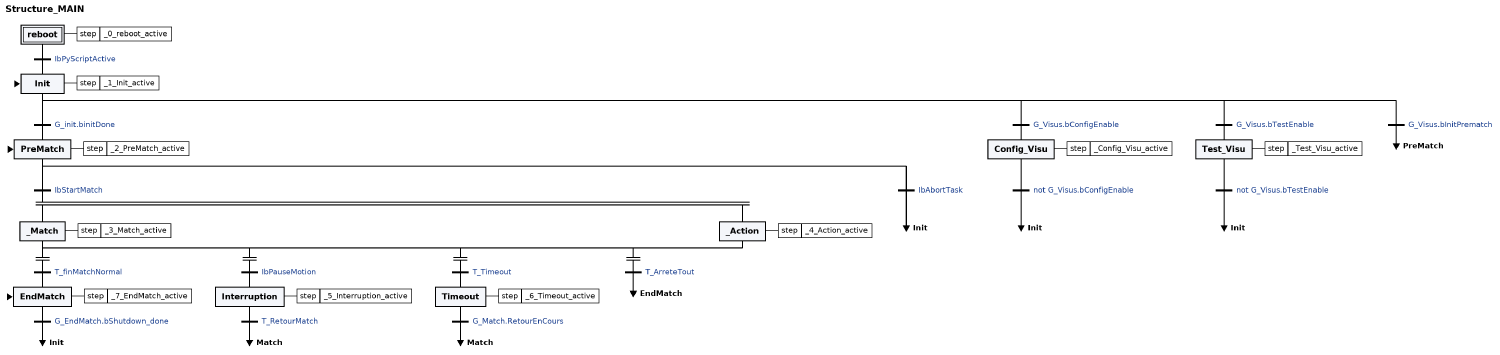
INITIAL_STEP reboot:
    _0_reboot_active(N);  // step action
END_STEP
TRANSITION FROM reboot TO Init
    := IbPyScriptActive;
END_TRANSITION
STEP Init:
    _1_Init_active(N);  // step action
END_STEP
TRANSITION FROM Init TO PreMatch
    := G_init.binitDone;
END_TRANSITION
TRANSITION FROM Init TO Config_Visu
    := G_Visus.bConfigEnable;
END_TRANSITION
STEP Config_Visu:
    _Config_Visu_active(N);  // step action
END_STEP
TRANSITION FROM Config_Visu TO Init
    := not G_Visus.bConfigEnable;
END_TRANSITION
TRANSITION FROM Init TO Test_Visu
    := G_Visus.bTestEnable;
END_TRANSITION
STEP Test_Visu:
    _Test_Visu_active(N);  // step action
END_STEP
TRANSITION FROM Test_Visu TO Init
    := not G_Visus.bTestEnable;
END_TRANSITION
TRANSITION FROM Init TO PreMatch
    := G_Visus.bInitPrematch;
END_TRANSITION
STEP PreMatch:
    _2_PreMatch_active(N);  // step action
END_STEP
TRANSITION FROM PreMatch TO (_Match, _Action)
    := IbStartMatch;
END_TRANSITION
TRANSITION FROM PreMatch TO Init
    := IbAbortTask;
END_TRANSITION
STEP _Match:
    _3_Match_active(N);  // step action
END_STEP
STEP _Action:
    _4_Action_active(N);  // step action
END_STEP
TRANSITION FROM (_Match, _Action) TO EndMatch
    := T_finMatchNormal;
END_TRANSITION
STEP EndMatch:
    _7_EndMatch_active(N);  // step action
END_STEP
TRANSITION FROM EndMatch TO Init
    := G_EndMatch.bShutdown_done;
END_TRANSITION
TRANSITION FROM (_Match, _Action) TO Interruption
    := IbPauseMotion;
END_TRANSITION
STEP Interruption:
    _5_Interruption_active(N);  // step action
END_STEP
TRANSITION FROM Interruption TO (_Match, _Action)
    := T_RetourMatch;
END_TRANSITION
TRANSITION FROM (_Match, _Action) TO Timeout
    := T_Timeout;
END_TRANSITION
STEP Timeout:
    _6_Timeout_active(N);  // step action
END_STEP
TRANSITION FROM Timeout TO (_Match, _Action)
    := G_Match.RetourEnCours;
END_TRANSITION
TRANSITION FROM (_Match, _Action) TO EndMatch
    := T_ArreteTout;
END_TRANSITION
// branch label Match

ACTION _0_reboot_active:
IF IbPyScriptActive THEN
	QbstartPyScript := FALSE;
ELSE
	QbstartPyScript := TRUE;
END_IF
END_ACTION

ACTION _1_Init_active:
IF IbAbortTask THEN
	G_init.ietapeInit := 0;
END_IF

CASE G_init.ietapeInit OF
	0://Mise à zéro et attende de l'ordre d'init
		QbstartBalise := FALSE;
		QbmoteurPower := FALSE;
		G_Prematch.bPrematchActive 	:= FALSE;
		G_EndMatch.bShutdown_done  	:= FALSE;
		G_Match.iLigne 				:= 0;
		IF IbStartInit THEN 
			G_init.ietapeInit := G_init.ietapeInit + 1;
		END_IF
	1://Mise sous tension des stepper moteurs de la base roulante (bloquage des roues)
		QbmoteurPower := TRUE;
		IF IbMoteurOn THEN
			G_init.ietapeInit := G_init.ietapeInit + 1;
			G_init.icounter := 1;
		END_IF;
	2://Activation du torque et des LED de tous les moteurs Dynamixels
		ITAction.DXLIN[G_init.icounter].bEnableTorque := TRUE;
		ITAction.DXLIN[G_init.icounter].bLedOn := TRUE;
		
		IF ITAction.DXLOUT[G_init.icounter].bEnableTorque AND ITAction.DXLOUT[G_init.icounter].bLedOn THEN 
			ITAction.DXLIN[G_init.icounter].bEnableTorque := FALSE;
			ITAction.DXLIN[G_init.icounter].bLedOn := FALSE;	
			G_init.icounter := G_init.icounter + 1;
		END_IF
		
		IF G_init.icounter > IiNumDynamixel THEN 
			G_init.ietapeInit := G_init.ietapeInit + 1;
		END_IF
		
	ELSE //Passage au prematch
		IF G_Visus.bInitPrematch OR G_Visus.bConfigEnable THEN 
			G_init.binitDone := TRUE;
			G_init.ietapeInit := 0;
		END_IF;
END_CASE

//à définir le nombre d'étape total pour que la visu affiche l'avancement sur une barre de progression
G_init.iNombreEtapeInit := 3;
G_Visus.iInitProgressBar := REAL_TO_INT(INT_TO_REAL(G_init.ietapeInit) / INT_TO_REAL(G_init.iNombreEtapeInit) * 100.0);

//switch en mode Test
IF VisuElems.CURRENTVISU = 'V_Test' THEN
	G_Visus.bTestEnable := TRUE;
ELSE
	G_Visus.bTestEnable := FALSE;
END_IF
END_ACTION

ACTION _2_PreMatch_active:
CASE IiChoixParcours OF
	0:
		P_Tableau_Strategie_1(bChoixCote := IbChoixCote);
		G_Match.Tableau := P_Tableau_Strategie_1.Tableau;
	1:
		P_Tableau_Strategie_2(bChoixCote := IbChoixCote);
		G_Match.Tableau := P_Tableau_Strategie_2.Tableau;
END_CASE

G_init.binitDone 			:= FALSE;
G_Match.PointMatch 			:= 0;
QbstartBalise 				:= FALSE;
G_Prematch.bPrematchActive 	:= TRUE;
ITMotion.odometrie.M_init_coordonne(IbChoixCote);
END_ACTION

ACTION _3_Match_active:
VisuElems.CURRENTVISU := 'V_Match';
//______________________________________________________________________________________________________________________________________________
//
// Comptage du Temps du match
//______________________________________________________________________________________________________________________________________________
IF NOT G_Match.MatchEnCours THEN
	G_Prematch.bPrematchActive := FALSE;
	G_Match.MatchEnCours := TRUE;
	G_Match.TimeStartMatch := TIME();
	G_Match.TimeStartLigne := TIME();
END_IF
G_Match.TimeMatch := TIME() - G_Match.TimeStartMatch; 

//______________________________________________________________________________________________________________________________________________
//
// Interpretation du Tableau
//______________________________________________________________________________________________________________________________________________
CASE G_Match.Tableau[G_Match.iLigne].TypeTache OF 
	

	//Temporisation-----------------------------------------------------------------------------------------------------------------------------
	eAttendre:
		IF delay(G_Match.TimeStartLigne, G_Match.Tableau[G_Match.iLigne].tAttente_ms)	THEN //Ligne suivante
			G_Match.PointMatch := G_Match.PointMatch + G_Match.Tableau[G_Match.iLigne].uiAjoutPoints_pts;
			G_Match.NextLigne := TRUE;
		END_IF
		
	//Changement de la ligne du Tableau----------------------------------------------------------------------------------------------------------
	eChangementTache:
		FOR G_Match.iCounter := 1 TO 100 DO
			IF G_Match.Tableau[G_Match.iCounter].NomEtape = G_Match.Tableau[G_Match.iLigne].EtapeCible THEN
				G_Match.iLigne := G_Match.iCounter - 1;
				EXIT;
			END_IF
		END_FOR
		G_Match.NextLigne := TRUE;
	
	//Action du robot => se gère dans _4_Action_active-------------------------------------------------------------------------------------------
	eAction: 
		IF G_Match.bActionFinie THEN //Ligne suivante
			G_Match.PointMatch := G_Match.PointMatch + G_Match.Tableau[G_Match.iLigne].uiAjoutPoints_pts;
			G_Match.NextLigne := TRUE;
		END_IF;	
	
	//Deplacement du robot-----------------------------------------------------------------------------------------------------------------------
	eDeplacement: 
		G_Match.bExecuteDeplacement := TRUE;
		IF G_Match.bDeplacementFini THEN //Ligne suivante
			G_Match.PointMatch := G_Match.PointMatch + G_Match.Tableau[G_Match.iLigne].uiAjoutPoints_pts;
			G_Match.bExecuteDeplacement := FALSE;
			G_Match.NextLigne := TRUE;
		END_IF
		
		//Gère le type de déplacement-------------------------------------------------------------------------------------------------------------
		CASE G_Match.Tableau[G_Match.iLigne].TypeDeplacement OF
			eCoordonne: 
				ITMotion.odometrie.M_move_to_coordonne(
				x 			:= G_Match.Tableau[G_Match.iLigne].lrPositionX_mm,
				y 			:= G_Match.Tableau[G_Match.iLigne].lrPositionY_mm,
				lrSpeed 	:= G_Match.Tableau[G_Match.iLigne].lrVitesse_mms,
				bExecute 	:= G_Match.bExecuteDeplacement,
				bbackward	:= FALSE,
				bDone 		=> G_Match.bDeplacementFini);
								
			eMarcheArriereCoordonne:
				ITMotion.odometrie.M_move_to_coordonne(
				x 			:= G_Match.Tableau[G_Match.iLigne].lrPositionX_mm,
				y 			:= G_Match.Tableau[G_Match.iLigne].lrPositionY_mm,
				lrSpeed 	:= G_Match.Tableau[G_Match.iLigne].lrVitesse_mms,
				bExecute 	:= G_Match.bExecuteDeplacement,
				bbackward	:= TRUE,
				bDone 		=> G_Match.bDeplacementFini);
			
			eDistance: 
				ITMotion.odometrie.M_move_distance(
				lrDistance 	:= G_Match.Tableau[G_Match.iLigne].lrDistanceVoulu_mm,
				lrSpeed 	:= G_Match.Tableau[G_Match.iLigne].lrVitesse_mms,
				bExecute 	:= G_Match.bExecuteDeplacement,
				bDone 		=> G_Match.bDeplacementFini);
				
			eAngle:
				ITMotion.odometrie.M_move_rotation(
				lrAngle 	:= G_Match.Tableau[G_Match.iLigne].lrAngleVoulu_deg,
				lrSpeed 	:= G_Match.Tableau[G_Match.iLigne].lrVitesse_mms,
				bExecute 	:= G_Match.bExecuteDeplacement,
				bDone 		=> G_Match.bDeplacementFini); 
			
			eCourbe:
				ITMotion.odometrie.M_move_curve(
				LrRayon		:= G_Match.Tableau[G_Match.iLigne].lrRayonCourbe_mm,
				LrAngle 	:= G_Match.Tableau[G_Match.iLigne].lrAngleVoulu_deg,
				lrSpeed 	:= G_Match.Tableau[G_Match.iLigne].lrVitesse_mms,				
				bExecute 	:= G_Match.bExecuteDeplacement,
				bDone 		=> G_Match.bDeplacementFini);
		END_CASE
END_CASE

//______________________________________________________________________________________________________________________________________________
//
// Passe à la ligne suivante du Tableau
//______________________________________________________________________________________________________________________________________________
IF G_Match.NextLigne THEN 
	G_Match.bActionFinie := FALSE;
	G_Match.bDeplacementFini := FALSE;
	G_Match.NextLigne := FALSE;
	G_Match.TimeStartLigne := TIME();
	G_Match.iLigne := G_Match.iLigne + 1; 
END_IF

//______________________________________________________________________________________________________________________________________________
//
// Debug
//______________________________________________________________________________________________________________________________________________

//affiche le nom de l'étape en cours pour le debug
IF G_Match.Tableau[G_Match.iLigne].NomEtape = '' THEN 
	QbEtapeEnCours := INT_TO_STRING(G_Match.iLigne); 
ELSE 
	QbEtapeEnCours := G_Match.Tableau[G_Match.iLigne].NomEtape;
END_IF;
END_ACTION

ACTION _4_Action_active:
IF G_Match.Tableau[G_Match.iLigne].TypeTache = eAction OR G_MAtch.iAsyncAction <> '' THEN 
///////////////////////////////////////////////////////////////////////////////////////////////////////////////////
// GESTION DES ACTIONS 
///////////////////////////////////////////////////////////////////////////////////////////////////////////////////

	IF StartAction('Lampe 3s') THEN
		
		G_IO.bLEDInit := TRUE;
		
		IF delay(G_match.TimeStartLigne, T#3S) THEN
			G_IO.bLEDInit := FALSE;
			FinishAction(0);
		END_IF;
		
//__________________________________________________________________________________________________________________
///////////////////////////////////////////////////////////////////////////////////////////////////////////////////
	ELSIF StartAction('Dynamixel position 0') THEN
		F_DXL_Position(0,500,ITAction.MoteurXL1);
//__________________________________________________________________________________________________________________
///////////////////////////////////////////////////////////////////////////////////////////////////////////////////		
	ELSIF StartAction('Dynamixel position 4095') THEN
		CASE G_Match.iEtapeAction OF
			0:
				ITAction.DXLIN[ITAction.MoteurXL1].bPosition := TRUE;
				ITAction.DXLIN[ITAction.MoteurXL1].ParamPosition_DINT := 10000;
				ITAction.DXLIN[ITAction.MoteurXL1].ParamSpeed_INT := 500;
				IF ITAction.DXLOUT[ITAction.MoteurXL1].bPosition THEN
					ITAction.DXLIN[ITAction.MoteurXL1].bPosition := FALSE;
					FinishAction(1);
					Next();
				END_IF
			1:
				ITAction.DXLIN[ITAction.MoteurXL1].bGetPosition := TRUE;
				IF PlusOuMoins(ITAction.DXLOUT[ITAction.MoteurXL1].INFO_Position_dint, 10000, 15) THEN 
					ITAction.DXLIN[ITAction.MoteurXL1].bGetPosition := FALSE;
					FinishAction(0);
				END_IF
		END_CASE
		
//__________________________________________________________________________________________________________________
///////////////////////////////////////////////////////////////////////////////////////////////////////////////////		
	ELSIF StartAction('Dynamixel reset') THEN
		F_DXL_Reset(ITAction.MoteurXL2,1,baseTime);
		
		
//__________________________________________________________________________________________________________________
///////////////////////////////////////////////////////////////////////////////////////////////////////////////////		
//--> Insérer les templates à partir d'ici 


///////////////////////////////////////////////////////////////////////////////////////////////////////////////////
// END_ACTION 
///////////////////////////////////////////////////////////////////////////////////////////////////////////////////
	ELSE //si aucune actione ne correspond au tableau TO DO
		pass();
	END_IF
END_IF



///////////////////////////////////////////////////////////////////////////////////////////////////////////////////
// DOCUMENTATION
///////////////////////////////////////////////////////////////////////////////////////////////////////////////////
(*

StartAction(Nom := "Nom de l'action");

FinishAction (StartAsync := FALSE, StopAsync := FALSE);

Next();

delay(last_time := G_Match.TimeStartLigne, tempo := T#1s);

PlusOuMoins(	val1  := G_A.DXL[G_A.Template].InfoPosition_DINT,
				val2  := 4095,
				plage := 15);
				
pass();
*)


///////////////////////////////////////////////////////////////////////////////////////////////////////////////////
// TEMPLATES A CUSTOMISER
///////////////////////////////////////////////////////////////////////////////////////////////////////////////////
(*
___________________________________________________________________________________________________________________

-> ACTION SIMPLE

///////////////////////////////////////////////////////////////////////////////////////////////////////////////////
	ELSIF StartAction('Nom Action') THEN
	
		"TON ACTION"
	
		IF "FIN DE L'ACTION" THEN
			FinishAction(0,0);
		END_IF
____________________________________________________________________________________________________________________		
		
-> CASE POUR L'ACTION

